// TwinCAT 3 PLC project MoldingCooler
// Title: Molding Cooling Tunnel
// Company: D_WFinePack
// ProjectVersion: 1.1.0
// ProgramVersion: 3.1.4020.4
// libraries:
//   Tc2_EtherCAT, * (Beckhoff Automation GmbH)
//   Tc2_Standard, * (Beckhoff Automation GmbH)
//   Tc2_System, * (Beckhoff Automation GmbH)
//   Tc2_SystemCX, * (Beckhoff Automation GmbH)
//   Tc2_Utilities, * (Beckhoff Automation GmbH)
//   Tc3_Module, * (Beckhoff Automation GmbH)
//   TemplateCore, * (TemplateCore Creators)
// project tree:
//   DUTs/Constants/ udtConstantsTransactions.TcDUT
//   DUTs/Database/ udtDBChannel.TcDUT, udtDBInterface.TcDUT, udtDBStoreFault.TcDUT, udtDBTransact.TcDUT
//   DUTs/RecipeData/ udtRecipe.TcDUT
//   DUTs/ udtCmpBaseMain.TcDUT, udtCmpServo.TcDUT, udtCmpVFD.TcDUT, udtEthercatSlaveStatus.TcDUT, udtHourlyData.TcDUT, udtIWS_DataLogItems.TcDUT, udtVFDCommand.TcDUT, udtVFDStatus.TcDUT, udtYaskawaVFDCmd.TcDUT, udtYaskawaVFDStatus.TcDUT
//   GVLs/ Globals.TcGVL
//   / PlcTask.TcTTO
//   POUs/ FB_DBTransaction.TcPOU, FB_PID.TcPOU, FB_Sensor.TcPOU, GlobalConfig.TcPOU, GlobalLogic.TcPOU
//   POUs/Stn100/ Stn100_00_ModeControl.TcPOU, Stn100_01_HMI.TcPOU, Stn100_02_Stats.TcPOU, Stn100_10_Main.TcPOU, Stn100_20_CoolingConveyor.TcPOU, Stn100_30_VibratoryConveyor.TcPOU, Stn100_40_Vibrator.TcPOU
// real-time tasks:
//   TASK PlcTask: cycle T#10ms, priority 10, ADS port 350
// I/O:
//   DEVICE EtherCat Master (EtherCAT), AmsNetId 5.49.24.194.2.1
//     Term 12 (EK1200) [EK1200-5000 EtherCAT Power supply (2A E-Bus)]
//       Term 13 (EL6070-0033) [EL6070-0033 1Ch. Licence key terminal, individual licences]
//       Term 14 (EL1034) [EL1034 4Ch. Dig. Input 24V, potential-free, 10µs]
//       Term 16 (EL1034) [EL1034 4Ch. Dig. Input 24V, potential-free, 10µs]
//       Term 17 (EL1034) [EL1034 4Ch. Dig. Input 24V, potential-free, 10µs]
//       Term 18 (EL1034) [EL1034 4Ch. Dig. Input 24V, potential-free, 10µs]
//       Term 19 (EL2798) [EL2798 8Ch. Dig. Output 24V AC/DC, 2A, potential-free]
//       Term 20 (EL2798) [EL2798 8Ch. Dig. Output 24V AC/DC, 2A, potential-free]
//       Term 21 (EL3314-0010) [EL3314-0010 4Ch. Ana Input Thermocouple (TC), High Precision]
//       Term 21 (EL6652) [EL6652 EtherNet/IP Scanner (Master)]
//       Term 23 (EK1110) [EK1110 EtherCAT extension]
//     Box 24 (Cooling Conv YASKAWA V1000 series) [YASKAWA V1000 series]
//     Box 25 (Vib Conv YASKAWA V1000 series) [YASKAWA V1000 series]
//     Box 26 (Vib Shaker YASKAWA V1000 series) [YASKAWA V1000 series]
//   DEVICE Device 2 (ECAT EIP Scanner (EL6652)), AmsNetId 5.49.24.194.3.1
//     Box 1 (FP7CPUS UNIT AFP7CPS31ES) // <INFO> </INFO> <EDS> 00D8000C00030100WN5.eds </EDS>
// variable links:
//   MoldingCooler/MoldingCooler Instance <-> Device 2 (ECAT EIP Scanner (EL6652))/Box 1 (FP7CPUS UNIT AFP7CPS31ES)
//     PlcTask Inputs/.gWeighRightCurrentRecipeID <-> Connection 2 (Input/Output)/Inputs/InByte_3
//     PlcTask Inputs/.gWeighRightInputs <-> Connection 2 (Input/Output)/Inputs/InByte
//   MoldingCooler/MoldingCooler Instance <-> EtherCat Master (EtherCAT)/Box 24 (Cooling Conv YASKAWA V1000 series)
//     PlcTask Inputs/Stn100_20_CoolingConveyor.iCurrentVelocity <-> Inputs_1/Output frequency
//     PlcTask Inputs/Stn100_20_CoolingConveyor.iStatus <-> Inputs/Drive status
//     PlcTask Outputs/Stn100_20_CoolingConveyor.oCommand <-> Outputs/Operation command
//     PlcTask Outputs/Stn100_20_CoolingConveyor.oSpeedReference <-> Outputs_1/Speed reference/limit
//   MoldingCooler/MoldingCooler Instance <-> EtherCat Master (EtherCAT)/Box 25 (Vib Conv YASKAWA V1000 series)
//     PlcTask Inputs/Stn100_30_VibratoryConveyor.iCurrentVelocity <-> Inputs_1/Output frequency
//     PlcTask Inputs/Stn100_30_VibratoryConveyor.iStatus <-> Inputs/Drive status
//     PlcTask Outputs/Stn100_30_VibratoryConveyor.oCommand <-> Outputs/Operation command
//     PlcTask Outputs/Stn100_30_VibratoryConveyor.oSpeedReference <-> Outputs_1/Speed reference/limit
//   MoldingCooler/MoldingCooler Instance <-> EtherCat Master (EtherCAT)/Box 26 (Vib Shaker YASKAWA V1000 series)
//     PlcTask Inputs/Stn100_40_Vibrator.iCurrentVelocity <-> Inputs_1/Output frequency
//     PlcTask Inputs/Stn100_40_Vibrator.iStatus <-> Inputs/Drive status
//     PlcTask Outputs/Stn100_40_Vibrator.oCommand <-> Outputs/Operation command
//     PlcTask Outputs/Stn100_40_Vibrator.oSpeedReference <-> Outputs_1/Speed reference/limit
//   MoldingCooler/MoldingCooler Instance <-> EtherCat Master (EtherCAT)/Term 12 (EK1200)/Term 14 (EL1034)
//     PlcTask Inputs/Stn100_00_ModeControl.iMovenCoolTankFull <-> Channel 2/Input
//     PlcTask Inputs/Stn100_10_Main.iBoxPres_Filling <-> Channel 4/Input
//     PlcTask Inputs/Stn100_10_Main.iWR_FillCmp <-> Channel 3/Input
//   MoldingCooler/MoldingCooler Instance <-> EtherCat Master (EtherCAT)/Term 12 (EK1200)/Term 16 (EL1034)
//     PlcTask Inputs/.iCycleStart <-> Channel 3/Input
//     PlcTask Inputs/.iCycleStop <-> Channel 4/Input
//   MoldingCooler/MoldingCooler Instance <-> EtherCat Master (EtherCAT)/Term 12 (EK1200)/Term 17 (EL1034)
//     PlcTask Inputs/Stn100_10_Main.iBoxPres_InfeedEntrance <-> Channel 1/Input
//     PlcTask Inputs/Stn100_10_Main.iBoxPres_Infeeed <-> Channel 2/Input
//     PlcTask Inputs/Stn100_10_Main.iBoxPres_OutFeed <-> Channel 3/Input
//     PlcTask Inputs/Stn100_10_Main.iBoxPres_OutFeedExit <-> Channel 4/Input
//   MoldingCooler/MoldingCooler Instance <-> EtherCat Master (EtherCAT)/Term 12 (EK1200)/Term 18 (EL1034)
//     PlcTask Inputs/Stn100_10_Main.iBoxCyl_DS_Retd <-> Channel 1/Input
//     PlcTask Inputs/Stn100_10_Main.iBoxCyl_US_Retd <-> Channel 2/Input
//   MoldingCooler/MoldingCooler Instance <-> EtherCat Master (EtherCAT)/Term 12 (EK1200)/Term 19 (EL2798)
//     PlcTask Outputs/Stn100_10_Main.oBoxCyl_DS_Ret <-> Channel 7/Output
//     PlcTask Outputs/Stn100_10_Main.oBoxCyl_US_Ret <-> Channel 8/Output
//     PlcTask Outputs/Stn100_10_Main.oInfeedConv_EntRelease <-> Channel 3/Output
//     PlcTask Outputs/Stn100_10_Main.oInfeedConv_Release <-> Channel 4/Output
//     PlcTask Outputs/Stn100_10_Main.oOutFeedConv_ExitRelease <-> Channel 6/Output
//     PlcTask Outputs/Stn100_10_Main.oOutFeedConv_Recieve <-> Channel 5/Output
//     PlcTask Outputs/Stn100_10_Main.oWeighRight_Ok2Fill <-> Channel 1/Output
//   MoldingCooler/MoldingCooler Instance <-> EtherCat Master (EtherCAT)/Term 12 (EK1200)/Term 20 (EL2798)
//     PlcTask Outputs/Stn100_00_ModeControl.oStackLightGreen <-> Channel 3/Output
//     PlcTask Outputs/Stn100_00_ModeControl.oStackLightHorn <-> Channel 4/Output
//     PlcTask Outputs/Stn100_00_ModeControl.oStackLightRed <-> Channel 1/Output
//     PlcTask Outputs/Stn100_00_ModeControl.oStackLightYellow <-> Channel 2/Output
//   MoldingCooler/MoldingCooler Instance <-> EtherCat Master (EtherCAT)/Term 12 (EK1200)/Term 21 (EL3314-0010)
//     PlcTask Inputs/Stn100_10_Main.iTempAtMoldDrop <-> TC Inputs Channel 1/Value
//     PlcTask Inputs/Stn100_10_Main.iTempAtShuteDrop <-> TC Inputs Channel 2/Value

CONFIGURATION MoldingCooler
    RESOURCE PLC ON TwinCAT3
        TASK PlcTask(INTERVAL := T#10ms, PRIORITY := 10);
        PROGRAM GlobalConfig WITH PlcTask : GlobalConfig;
        PROGRAM GlobalLogic WITH PlcTask : GlobalLogic;
        PROGRAM Stn100_00_ModeControl WITH PlcTask : Stn100_00_ModeControl;
        PROGRAM Stn100_01_HMI WITH PlcTask : Stn100_01_HMI;
        PROGRAM Stn100_02_Stats WITH PlcTask : Stn100_02_Stats;
        PROGRAM Stn100_10_Main WITH PlcTask : Stn100_10_Main;
        PROGRAM Stn100_20_CoolingConveyor WITH PlcTask : Stn100_20_CoolingConveyor;
        PROGRAM Stn100_30_VibratoryConveyor WITH PlcTask : Stn100_30_VibratoryConveyor;
        PROGRAM Stn100_40_Vibrator WITH PlcTask : Stn100_40_Vibrator;
    END_RESOURCE
END_CONFIGURATION

// ---- DUTs/Constants/udtConstantsTransactions.TcDUT
TYPE udtConstantsTransactions :
STRUCT
	FindSlot : INT := 1;
	GetAssignedStation: INT := 2;
	GetLineStatus : INT := 3;
	GetOrderData : INT := 4;
	GetPalletData: INT := 5;
	GetUnusedPalletID : INT := 6;
	SetOrderData : INT := 7;
	SetPalletData : INT := 8;
	StoreFault : INT := 9;
	GetAlignerData : INT := 10;
	DebugGetPartialAID : INT := 11;
	SetManualAID : INT :=12;
	DebugLookupAlignerInBatch :INT := 13;
	DebugAssignDummyAligner :INT := 14;
END_STRUCT
END_TYPE

// ---- DUTs/Database/udtDBChannel.TcDUT
TYPE udtDBChannel :
STRUCT
	CurrentUser:DINT;
	ErrorCode: DINT;
	ErrorMessage: STRING[256];
	DataIn: ARRAY[0..1999] OF BYTE;
	DataOut: ARRAY[0..1999] OF BYTE;
END_STRUCT
END_TYPE

// ---- DUTs/Database/udtDBInterface.TcDUT
TYPE udtDBInterface :
STRUCT
	Trigger: DWORD;
	Response: DWORD;
	Lock: BOOL;
	Connection: ARRAY[0..19] OF udtDBChannel;
END_STRUCT
END_TYPE

// ---- DUTs/Database/udtDBStoreFault.TcDUT
TYPE udtDBStoreFault :
STRUCT
	Station : DINT;
	FaultCode: DINT;
	FaultText : STRING[255];
	AcknowledgeTime: REAL;
	Duration: REAL;
	TimeStamp:Timestamp;
	Data1 : REAL;
	Data2 : REAL;
	Data3:  REAL;
	StringData1 : STRING[255];
	StringData2 : STRING[255];
	ResultCode: DINT;
	ResultText: STRING[255] ;
END_STRUCT
END_TYPE

// ---- DUTs/Database/udtDBTransact.TcDUT
TYPE udtDBTransact :
STRUCT
	Start: BOOL;
	Done: BOOL;
	ErrorCode: DINT;
	ErrorMessage : STRING[256];
	pDatabaseInterface: POINTER TO udtDBInterface;
	UserID: DINT;
	TransactionID: INT;
	DataLength: DINT;
	DataOutLength: DINT;
	DataIn: ARRAY[0..1999] OF BYTE;
	DataOut: ARRAY[0..1999] OF BYTE;
	State: DINT;
END_STRUCT
END_TYPE

// ---- DUTs/RecipeData/udtRecipe.TcDUT
TYPE udtRecipe :
STRUCT
	Matnr: STRING;
	Maktx: STRING;
	Pic_Name: STRING;
	VisionID: DINT;
	nBatchID: DINT;
	QuantityToProduce: DINT;
	Remaining: DINT;
	LoadConv_Speed: REAL;
	HopperElev_Speed: REAL;
	SeparatorConv_Speed: REAL;
	PaddleWheel_Speed: REAL;
	SortingConv_Speed: REAL;
	Wrapper_Speed: REAL;
	Wrapper_TempSP: REAL;
	Wrapper_VacuumSP: REAL;
END_STRUCT
END_TYPE

// ---- DUTs/udtCmpBaseMain.TcDUT
TYPE udtCmpBaseMain :
STRUCT
	Framework: Framework;
END_STRUCT
END_TYPE

// ---- DUTs/udtCmpServo.TcDUT
TYPE udtCmpServo :
STRUCT
	Framework: Framework;
	BaseSpeedRef: REAL;
	RunReq: BOOL;
	Running: BOOL;
END_STRUCT
END_TYPE

// ---- DUTs/udtCmpVFD.TcDUT
TYPE udtCmpVFD :
STRUCT
	Framework: Framework;
	BaseSpeedRef: REAL;
	RunReq: BOOL;
	Running: BOOL;
END_STRUCT
END_TYPE

// ---- DUTs/udtEthercatSlaveStatus.TcDUT
TYPE udtEthercatSlaveStatus :
STRUCT
	Address : WORD;
	Name : STRING[31];
	DeviceState: BYTE;
	LinkState: BYTE;
	SlaveStateBits: ST_EcSlaveStateBits;
END_STRUCT
END_TYPE

// ---- DUTs/udtHourlyData.TcDUT
TYPE udtHourlyData :
STRUCT
	GoodCount :DINT :=0;
	ScrapCount :DINT :=0;	
END_STRUCT
END_TYPE

// ---- DUTs/udtIWS_DataLogItems.TcDUT
TYPE udtIWS_DataLogItems :
STRUCT
	HourlyTranReq :BOOL  :=0;
	HourlyTranCmp :BOOL  :=0;
	CurrOeeTranReq :BOOL  :=0;
	CurrOeeTranCmp :BOOL  :=0;
	ShiftOeeTranReq :BOOL  :=0;
	ShiftOeeTranCmp :BOOL  :=0;
	FaultedTranReq :BOOL  :=0;
	FaultedTranCmp :BOOL  :=0;
	FailureTranReq :BOOL  :=0;
	FailureTranCmp :BOOL  :=0;
	CreateNewBatchReq :BOOL  :=0;
	CreateNewBatchCmp :BOOL  :=0;
END_STRUCT
END_TYPE

// ---- DUTs/udtVFDCommand.TcDUT
TYPE udtVFDCommand :
STRUCT
	Stop : BOOL;
	Start: BOOL;
	Jog: BOOL;
	ClearFaults: BOOL;
	RunFwd: BOOL;
	RunRev: BOOL;
	ForceKeypadCtrl: BOOL;
	MOPIncrement: BOOL;
	AccelRate1: BOOL;
	AccelRate2: BOOL;
	DecelRate1: BOOL;
	DecelRate2: BOOL;
	FreqSel01: BOOL;
	FreqSel02: BOOL;
	FreqSel03: BOOL;
	MOPDecrement: BOOL;
END_STRUCT
END_TYPE

// ---- DUTs/udtVFDStatus.TcDUT
TYPE udtVFDStatus :
STRUCT
	Ready : BOOL;
	Active: BOOL;
	CommandFwd: BOOL;
	RunningFwd: BOOL;
	Accelerating: BOOL;
	Decelerating: BOOL;
	Reserved: BOOL;	
	Faulted: BOOL;
	AtSpeed: BOOL;
	CommFreqCnt: BOOL;
	CommLogicCnt: BOOL;
	ParmsLocked: BOOL;
	DigIn1Active: BOOL;
	DigIn2Active: BOOL;
	DigIn3Active: BOOL;
	DigIn4Active: BOOL;
END_STRUCT
END_TYPE

// ---- DUTs/udtYaskawaVFDCmd.TcDUT
TYPE udtYaskawaVFDCmd :
STRUCT
	RunFwd :BOOL;
	RunRev :BOOL;
	ClearFaults :BOOL;	
END_STRUCT
END_TYPE

// ---- DUTs/udtYaskawaVFDStatus.TcDUT
TYPE udtYaskawaVFDStatus :
STRUCT
Running :BOOL;	
ZeroSpeed :BOOL;
RunningFWD :BOOL;
SpeedAgree :BOOL;
Ready :BOOL;
Alarm :BOOL;
Faulted :BOOL;
OpError :BOOL;
PowerLoss:BOOL;
END_STRUCT
END_TYPE

// ---- GVLs/Globals.TcGVL
{attribute 'Tc2GvlVarNames'}
{attribute 'qualified_only'}
VAR_GLOBAL
	(*Wired Inputs for Station Control*)
	iCycleStart AT %I* :BOOL;
	iCycleStop AT %I* :BOOL;
	
	gDatabaseInterface: udtDBInterface;
	gInitialScanForce: BOOL:=0;
	gFirstScan: BOOL:=0;
	gTimeZoneOffsetFromUTC: DINT;
	gCurrentTime: timestamp;
	gSoftwareRevision : STRING;
	gDbTransact :ARRAY[0..1] OF udtIWS_DataLogItems;
	
	(*Create the Hourly Containers*)
	gCurrShift :DINT;
	gLastShift :DINT;
	gCurrentHour :DINT;
	gLastHour : DINT;
	gTargetRatePerHour : DINT;
	gTargetRatePerMin : DINT;
	gRejectRate : REAL;
	gHourlyData: ARRAY[0..23] OF udtHourlyData;
	gShiftdata :ARRAY[0..3] OF udtHourlyData;
	gCurrOeeLogTime :TIME := T#300000MS;
	

	(*Station 100*)
	gStation100: Station;
	gStn100_02_Stats : Component_Stats;
	gStn100_StateTraceBuffer : TraceFIFOBuffer;
	gStn100_StateTraceFifo : FIFO_StateTrace := ( Overwrite := TRUE );
	gStn100_HMIMessageBuffer : HMIMessageBuffer;
	gStn100_HMIMessageFIFO : FIFO_HMIMessage := (Overwrite := TRUE);
	gStn100_10_Main : udtCmpBaseMain;
	gStn100_20_CoolingConveyor : udtCmpVFD;
	gStn100_30_VibratoryConveyor : udtCmpVFD;
	gStn100_40_Vibrator : udtCmpVFD;
	gStn100FaultedNotAck: BOOL;	
	
	(* Ethernet IP Inputs from Weigh Scale *)
		gWeighRightInputs AT %I* : INT;
		gWeighRightCurrentRecipeID AT %I* :INT;

END_VAR

VAR_GLOBAL PERSISTENT
	gCurrProduct : udtRecipe;
END_VAR

VAR_GLOBAL CONSTANT
	strNull : STRING :='';
	cStats: StatsConstants;
	gstLibVersion : ST_LibVersion;
END_VAR

// ---- POUs/GlobalConfig.TcPOU
PROGRAM GlobalConfig
VAR
	FirstScan:R_TRIG;
	FBStartHMI:NT_StartProcess;
	tmrDelayHMIStart:TON;

	fbNTGetLocalTime : FB_LocalSystemTime;
	LocalSystemTime : T_FileTime;
	fbDisplay : FB_CXSetTextDisplay;
	hiStartOfShift1Min : DINT;
	hiStartOfShift1Hour : DINT;
	hiStartOfShift2Min : DINT;
	hiStartOfShift2Hour : DINT;
	hiStartOfShift3Min : DINT;
	hiStartOfShift3Hour : DINT;
	hiPlannedDownTimeShift1Min : DINT;
	hiPlannedDownTimeShift2Min : DINT;
	hiPlannedDownTimeShift3Min : DINT;
	hiIdealCycleTime : REAL;
	hiAggregateInterval : DINT;
	TempFullRate : DINT;
	TempRateCalc : FLOAT;
	tempRejectRate : FLOAT;
	
	tTime : TimeStamp;
	END_VAR

FirstScan(CLK:=TRUE);
Globals.gFirstScan:=FirstScan.Q OR Globals.gInitialScanForce;
Globals.gInitialScanForce := FALSE;
IF Globals.gFirstScan THEN
	(*Initialize all FIFOs to avoid Access Violation exception*)
	Globals.gStn100_StateTraceFifo.INIT(pFIFO := ADR(Globals.gStn100_StateTraceBuffer));
	Globals.gStation100.AttentionRequiredFIFO.INIT(pFIFO := ADR(Globals.gStation100.AttentionRequiredFIFOBuffer));
	Globals.gStation100.NotOKtoStopFIFO.INIT(pFIFO := ADR(Globals.gStation100.NotOKToStopFIFOBuffer));
	Globals.gStation100.FaultedFIFO.INIT(pFIFO := ADR(Globals.gStation100.FaultedFIFOBuffer));
	Globals.gStation100.HMIMessageFIFO.INIT(pFIFO := ADR(Globals.gStation100.HMIMessageBuffer));
	
	(*Set Time Zone*)
	Globals.gTimeZoneOffsetFromUTC := -7;
	Globals.gSoftwareRevision := Dint_to_String(Globals.gstLibVersion.iRevision);
	Globals.gStation100.MachineID :=4;
	
	(*Set Initial Start Of Shift Values HackAlert*)
	Globals.gStn100_02_Stats.StartOfShift[0,0] :=0;	
	Globals.gStn100_02_Stats.StartOfShift[0,1] :=7;	
	Globals.gStn100_02_Stats.StartOfShift[1,0] :=0;	
	Globals.gStn100_02_Stats.StartOfShift[1,1] :=15;	
	Globals.gStn100_02_Stats.StartOfShift[2,0] :=0;	
	Globals.gStn100_02_Stats.StartOfShift[2,1] :=23;		
END_IF

(*Set display*)
fbDisplay(bExecute := Globals.gFirstScan,
			nDevID := 2,
			nMode := e_CX1100_WRITELine1,
			stLine := 'DW2164_rev01',
			nCursorPos := 0);

fbNTGetLocalTime(
	sNetID:='' ,
	bEnable:= TRUE,
	dwCycle:= 1,
	dwOpt:= 0,
	tTimeout:= DEFAULT_ADS_TIMEOUT );
LocalSystemTime := SYSTEMTIME_TO_FILETIME(fbNTGetLocalTime.systemTime);
Globals.gCurrentTime.CurrentValue.dwHighPart := LocalSystemTime.dwHighDateTime;
Globals.gCurrentTime.CurrentValue.dwLowPart := LocalSystemTime.dwLowDateTime;
Globals.gCurrentTime.DateTime := fbNTGetLocalTime.systemTime;
templatecore.GVL.gCurrentTime := Globals.gCurrentTime;

tTime := Globals.gCurrentTime;
tempRejectRate := (Globals.gRejectRate / 1000);
TempFullRate :=(Globals.gTargetRatePerMin*60);
TempRateCalc := FLOAT_TO_DINT(TempFullRate*(tempRejectRate));
Globals.gTargetRatePerHour := (TempFullRate-FLOAT_TO_DINT(TempRateCalc));

(*STATION 100*)
(*Reset logic for top-level main component*)
Globals.gStn100_10_Main.Framework.ResetStart := Globals.gStation100.CycleReset;
IF Globals.gStn100_10_Main.Framework.ResetDone THEN
	Globals.gStation100.ResetDone := TRUE;
ELSE
	Globals.gStation100.ResetDone := FALSE;
END_IF

(*Set Component IDs and Configurations*)
Globals.gStation100.StationID := 100;
Globals.gStn100_02_Stats.Framework.ComponentIDRecord.ID := 2;
Globals.gStn100_02_Stats.Framework.ComponentIDRecord.Name := 'Stats';
Globals.gStn100_10_Main.Framework.ComponentIDRecord.ID := 10;
Globals.gStn100_10_Main.Framework.ComponentIDRecord.Name := 'Main';
Globals.gStn100_20_CoolingConveyor.Framework.ComponentIDRecord.ID := 20;
Globals.gStn100_20_CoolingConveyor.Framework.ComponentIDRecord.Name := 'Cooling Conv';
Globals.gStn100_30_VibratoryConveyor.Framework.ComponentIDRecord.ID := 30;
Globals.gStn100_30_VibratoryConveyor.Framework.ComponentIDRecord.Name := 'Vibratory Conv';
Globals.gStn100_40_Vibrator.Framework.ComponentIDRecord.ID := 40;
Globals.gStn100_40_Vibrator.Framework.ComponentIDRecord.Name := 'Vibrator';


IF Globals.gStn100_02_Stats.IdealCycleTime <= 0.3 THEN
	Globals.gStn100_02_Stats.IdealCycleTime := 0.3; (*time in seconds*)
END_IF
Globals.gStn100_02_Stats.AggregateInterval := 3; (*aggregate time in minutes*)
IF Globals.gStn100_02_Stats.AggregateInterval < 1 THEN
	Globals.gStn100_02_Stats.AggregateInterval  := 1;
END_IF

(*Handle The HMI OEE Config Items*)
IF ((NOT Globals.gStation100.CycleAuto) AND (NOT Globals.gStation100.CycleFaulted)) THEN
	IF (hiStartOfShift1Min >0 AND hiStartOfShift1Min <> Globals.gStn100_02_Stats.StartOfShift[0,0]) THEN
		Globals.gStn100_02_Stats.StartOfShift[0,0] := hiStartOfShift1Min;
	END_IF
	IF (hiStartOfShift1Hour >0 AND hiStartOfShift1Hour <> Globals.gStn100_02_Stats.StartOfShift[0,1]) THEN
		Globals.gStn100_02_Stats.StartOfShift[0,1] := hiStartOfShift1Hour;
	END_IF
	IF (hiStartOfShift2Min >0 AND hiStartOfShift2Min <> Globals.gStn100_02_Stats.StartOfShift[1,0]) THEN
		Globals.gStn100_02_Stats.StartOfShift[1,0] := hiStartOfShift2Min;
	END_IF	
	IF (hiStartOfShift2Hour >0 AND hiStartOfShift2Hour <> Globals.gStn100_02_Stats.StartOfShift[1,1]) THEN
		Globals.gStn100_02_Stats.StartOfShift[1,1] := hiStartOfShift2Hour;
	END_IF	
	IF (hiStartOfShift3Min >0 AND hiStartOfShift3Min <> Globals.gStn100_02_Stats.StartOfShift[2,0]) THEN
		Globals.gStn100_02_Stats.StartOfShift[2,0] := hiStartOfShift3Min;
	END_IF	
	IF (hiStartOfShift3Hour >0 AND hiStartOfShift3Hour <> Globals.gStn100_02_Stats.StartOfShift[2,1]) THEN
		Globals.gStn100_02_Stats.StartOfShift[2,1] := hiStartOfShift3Hour;
	END_IF	
	IF (hiPlannedDownTimeShift1Min >0 AND hiPlannedDownTimeShift1Min <> Globals.gStn100_02_Stats.PlannedDownTime[0]) THEN
		Globals.gStn100_02_Stats.PlannedDownTime[0] := hiPlannedDownTimeShift1Min;
	END_IF	
	IF (hiPlannedDownTimeShift2Min >0 AND hiPlannedDownTimeShift2Min <> Globals.gStn100_02_Stats.PlannedDownTime[1]) THEN
		Globals.gStn100_02_Stats.PlannedDownTime[1] := hiPlannedDownTimeShift2Min;
	END_IF	
	IF (hiPlannedDownTimeShift3Min >0 AND hiPlannedDownTimeShift3Min <> Globals.gStn100_02_Stats.PlannedDownTime[2]) THEN
		Globals.gStn100_02_Stats.PlannedDownTime[2] := hiPlannedDownTimeShift3Min;
	END_IF		
	IF (hiIdealCycleTime >0 AND hiIdealCycleTime <> Globals.gStn100_02_Stats.IdealCycleTime) THEN
		Globals.gStn100_02_Stats.IdealCycleTime := hiIdealCycleTime;
	END_IF	
	IF (hiAggregateInterval >0 AND hiAggregateInterval <> Globals.gStn100_02_Stats.AggregateInterval) THEN
		Globals.gStn100_02_Stats.AggregateInterval := hiAggregateInterval;
	END_IF	
END_IF

END_PROGRAM

// ---- POUs/GlobalLogic.TcPOU
PROGRAM GlobalLogic
VAR
	(*Create the Objects for Data Collection of Rates*)
	hiHourDataLogReq :BOOL :=0;
	hoHourDataLogAck :BOOL :=0;	
	hiShiftDataLogReq :BOOL :=0;
	hoShiftDataLogAck :BOOL :=0;
	hiCurrOeeLogReq  :BOOL :=0;
	hoCurrOeeLogAck  :BOOL :=0;	
	hiShiftOeeLogReq  :BOOL :=0;
	hoShiftOeeLogAck  :BOOL :=0;		

	State :DINT :=0;
	NextState :DINT :=0;
	FirstEntry: BOOL;
	tmrState: TON;	
	tmrState20 :TON;
	tmrState40 :TON;
	tmrState50 :TON;
	tmrState70 :TON;
	tmrState80 :TON;
	tmrState100 :TON;
	tmrState110 :TON;
	tmrCurrOeeLog :TON;	
END_VAR

IF Globals.gFirstScan THEN
	tmrCurrOeeLog(in:=TRUE,pt:=Globals.gCurrOeeLogTime);
END_IF

(*Set HMI Flags for the Requested Data Log Event*)
IF (Globals.gCurrShift <> Globals.gLastShift) THEN
	hiShiftDataLogReq :=TRUE;	
END_IF

IF (Globals.gCurrentHour <> Globals.gLastHour) THEN
	hiHourDataLogReq :=TRUE;	
END_IF
tmrCurrOeeLog(in:=TRUE);
IF (tmrCurrOeeLog.Q) THEN	
	hiCurrOeeLogReq :=TRUE;
END_IF

IF NextState <> State THEN
	(*code: Log state change into buffer*)
	FirstEntry := TRUE;
	State := NextState;
ELSE
	FirstEntry := FALSE;
END_IF

IF FirstEntry THEN
	tmrState(IN:=FALSE);
	tmrState20(IN:=FALSE);
	tmrState40(IN:=FALSE);
	tmrState50(IN:=FALSE);
	tmrState70(IN:=FALSE);
	tmrState80(IN:=FALSE);	
	tmrState100(IN:=FALSE);
	tmrState110(IN:=FALSE);	
END_IF

CASE State OF
	
0:	(*Check If we have any Data logging Requests *)
		IF (hiHourDataLogReq)OR(Globals.gDbTransact[0].HourlyTranReq AND Globals.gDbTransact[0].HourlyTranCmp) THEN
			Globals.gDbTransact[0].HourlyTranReq := TRUE;
			NextState:=10;
		END_IF
		IF (hiShiftDataLogReq)OR (Globals.gDbTransact[0].ShiftOeeTranReq AND Globals.gDbTransact[0].ShiftOeeTranCmp) THEN
			Globals.gDbTransact[0].ShiftOeeTranReq := TRUE;
			NextState:=40;
		END_IF	
		IF (hiCurrOeeLogReq) THEN
			Globals.gDbTransact[0].CurrOeeTranReq := TRUE;
			NextState:=70;
		END_IF
(*		IF (hiShiftOeeLogReq) THEN
			Globals.gDbTransact[0].ShiftOeeTranReq := TRUE;			
			NextState:=100;
		END_IF *)

10:	(*Wait for confirmation from HMI For Hourly data Logging*)

	tmrState(IN:=TRUE, PT:=T#3.0S);
	hoHourDataLogAck := (Globals.gDbTransact[0].HourlyTranReq AND Globals.gDbTransact[0].HourlyTranCmp);
	IF hoHourDataLogAck THEN
		NextState:=20;
		Globals.gDbTransact[0].HourlyTranReq := FALSE;
		Globals.gDbTransact[0].HourlyTranCmp := FALSE;
	END_IF
	IF  tmrState.Q THEN
		hiHourDataLogReq := FALSE;
		hoHourDataLogAck := FALSE;
		Globals.gDbTransact[0].HourlyTranReq := FALSE;
		Globals.gDbTransact[0].HourlyTranCmp := FALSE;
		NextState:=0;
	END_IF

20:	(*Clear Hour DataLogging Events*)
	hoHourDataLogAck := (Globals.gDbTransact[0].HourlyTranReq AND Globals.gDbTransact[0].HourlyTranCmp);
	tmrState20(IN:=TRUE, PT:=T#3.0S);
	IF NOT hoHourDataLogAck AND NOT tmrState.Q THEN
		Globals.gLastHour := Globals.gCurrentHour ;
		Globals.gHourlyData[Globals.gCurrentHour].GoodCount :=0;
		Globals.gHourlyData[Globals.gCurrentHour].ScrapCount :=0;
		NextState:=0;		
	END_IF
	IF  tmrState20.Q THEN
		hiHourDataLogReq := TRUE;
		hoHourDataLogAck := FALSE;
		NextState:=0;
	END_IF
	
40:	(*Wait for confirmation from HMI For Shift data Logging*)
	hoShiftDataLogAck :=(Globals.gDbTransact[0].ShiftOeeTranReq AND Globals.gDbTransact[0].ShiftOeeTranCmp);
	tmrState40(IN:=TRUE, PT:=T#3.0S);
	IF hoShiftDataLogAck THEN
		NextState:=50;
		Globals.gDbTransact[0].ShiftOeeTranReq := FALSE;
		Globals.gDbTransact[0].ShiftOeeTranCmp := FALSE;
	END_IF
	IF  tmrState40.Q THEN
		hiShiftDataLogReq := FALSE;
		hoShiftDataLogAck := FALSE;
		NextState:=0;
	END_IF

50:	(*Clear Shift data Logging Event*)
	hoShiftDataLogAck :=(Globals.gDbTransact[0].ShiftOeeTranReq AND Globals.gDbTransact[0].ShiftOeeTranCmp);
	tmrState50(IN:=TRUE, PT:=T#3.0S);
	IF NOT hoHourDataLogAck THEN
		Globals.gLastShift := Globals.gCurrShift;
		(*Globals.gShiftData[Globals.gCurrShift].GoodCount :=0;
		Globals.gShiftData[Globals.gCurrShift].ScrapCount :=0;
		MEMSET(ADR(Stn100_02_Stats.DBShiftOeeRecord),0,SIZEOF(Stn100_02_Stats.DBShiftOeeRecord)); *)
		hiShiftOeeLogReq :=FALSE;			
		NextState:=0;	
	END_IF
	IF  tmrState50.Q THEN
		hiShiftDataLogReq := TRUE;
		hoShiftDataLogAck := FALSE;
		NextState:=0;
	END_IF	

70:	(*Wait for confirmation from HMI For Current OEE Data Logging*)
	hoCurrOeeLogAck :=(Globals.gDbTransact[0].CurrOeeTranReq AND Globals.gDbTransact[0].CurrOeeTranCmp);
	tmrState70(IN:=TRUE, PT:=T#3.0S);
	IF hoCurrOeeLogAck OR tmrState70.Q THEN
		NextState:=80;
		tmrCurrOeeLog(IN:=FALSE);
		Globals.gDbTransact[0].CurrOeeTranReq := FALSE;
		Globals.gDbTransact[0].CurrOeeTranCmp := FALSE;
	END_IF
	IF  tmrState70.Q THEN
		hiCurrOeeLogReq := FALSE;
		hoCurrOeeLogAck := FALSE;
		tmrCurrOeeLog(IN:=TRUE);		
		NextState:=0;
	END_IF

80:	(*Clear Current Oee Data Logging Event*)
	hoCurrOeeLogAck :=(Globals.gDbTransact[0].CurrOeeTranReq AND Globals.gDbTransact[0].CurrOeeTranCmp);
	tmrState80(IN:=TRUE, PT:=T#3.0S);
	IF NOT hoCurrOeeLogAck THEN
		NextState :=0;
	END_IF
	
	IF  tmrState80.Q THEN
		hiCurrOeeLogReq := TRUE;
		hoCurrOeeLogAck := FALSE;
		Globals.gDbTransact[0].CurrOeeTranReq := FALSE;
		Globals.gDbTransact[0].CurrOeeTranCmp := FALSE;
		NextState:=0;
	END_IF	
	
100: (*Wait for confirmation from HMI For Shift OEE Data Logging*)
	tmrState100(IN:=TRUE, PT:=T#3.0S);
	IF hoShiftOeeLogAck OR tmrState100.Q THEN
		NextState:=110;
	END_IF
	IF  tmrState100.Q THEN
		hiShiftOeeLogReq := FALSE;
		hoShiftOeeLogAck := FALSE;
		NextState:=0;
	END_IF

110: (*Clear*)
	tmrState110(IN:=TRUE, PT:=T#3.0S);
	IF NOT hoShiftOeeLogAck THEN
		NextState :=0;
	END_IF
	
	IF  tmrState110.Q THEN
		hiShiftOeeLogReq := FALSE;
		hoShiftOeeLogAck := FALSE;
		NextState:=0;
	END_IF		
	
END_CASE

END_PROGRAM

// ---- POUs/Stn100/Stn100_00_ModeControl.TcPOU
PROGRAM Stn100_00_ModeControl
VAR
	pStation: POINTER TO Station;
	pMain: POINTER TO udtCmpBaseMain;
	Local: FrameworkLocal;
	tmrDelayPCStart: TON;
	tmrWritePersistentData: TON;
	tmrWritePersistentDataPulse: TON;
	fbStartPC: NT_StartProcess;
	fbGetTime: GETSYSTEMTIME;
	fbWritePersistentData: FB_WritePersistentData;
	StationResetRequest: BOOL;
	MsgText: STRING256;
	AltMsgText: STRING256;
	FaultText: STRING256;
	FaultAltText: STRING256;
	FaultNumber: INT;
	FaultData: StatsFault;
	StationLevelFault: BOOL;
	TempEvent: StatsEvent;
	TimeStamp: StateTimeStamp;
	CurrentTime: TIMESTRUCT;
	TimeLo: UDINT;
	TimeHi: UDINT;
	cmdStart: BOOL;
	cmdOperatorStop: BOOL;
	cmdMachineStop: BOOL;
	cmdFaultAcknowledge: BOOL;
	cmdFullInit: BOOL;
	cmdFaultReset: BOOL;
	cmdSingleStepOn: BOOL;
	cmdSingleStepOff: BOOL;
	cmdSingleStepAdvance: BOOL;
	cmdManualMode: BOOL;
	OKToStart: BOOL;
	OKToReset: BOOL;
	onsStart: R_TRIG;
	onsOperatorStop: R_TRIG;
	onsMachineStop: R_TRIG;
	onsFaultAcknowledge: R_TRIG;
	onsStationReset: R_TRIG;
	onsFaultReset: R_TRIG;
	onsSingleStepOn: R_TRIG;
	onsSingleStepOff: R_TRIG;
	onsSingleStepAdvance: R_TRIG;
	onsManualMode: R_TRIG;
	onsEStopNotOKHMIMessage: BOOL;
	onsEStopNotOKStartAttmpt: BOOL;
	onsPowerOnAttmpt: BOOL;
	onsAirNotOKHMIMessage: BOOL;
	onsAirNotOKStartAttempt: BOOL;
	onsEStopSafetyEDMErrorHMIMessage: BOOL;
	onsEStopSafetyEDMErrorStartAttempt: BOOL;
	onsGateSafetyEDMErrorHMIMessage: BOOL;
	onsGateSafetyEDMErrorStartAttempt: BOOL;
	onsSortingConvSafetyEDMErrorHMIMessage: BOOL;
	onsSortingConvSafetyEDMErrorStartAttempt: BOOL;
	onsCrossConvSafetyEDMErrorHMIMessage: BOOL;
	onsCrossConvSafetyEDMErrorStartAttempt: BOOL;	
	onsGateNotLockedHMIMessage: BOOL;
	onsPrematureStartAttempt: BOOL;
	onsStartAttemptBeforePreheat: BOOL;
	WaitForResetMsg: BOOL;
	SeparateAckAndReset: BOOL := TRUE;
	bStartingToRun: BOOL;
	b500msPulse: BOOL;
	tmrPulseON: TON;
	tmrPulseOFF: TON;
	tmrState: TON;
	tmrControlPowerPBPressedDelay: TON;
	tmrAirPressureNotOK: TON;
	tmrMoveNCoolTankNotOK: TON;
	tmrOKToStop: TON;
	tmrGateLock: TON;
	cColor: Colors;
	cChannel: Channels;
	cStats: StatsConstants;	
	
	(*Inputs*)
	iEStopOK :BOOL;
	iEStopGateOK: BOOL;
	iEstopMainEnclosurePBReleased: BOOL;
	iEstopGatePBReleased: BOOL;
	iEstopRobotPBReleased: BOOL;
	iEstopGateClosed: BOOL;
	iEstopWrapperPBReleased: BOOL;
	iEstopWrapperGateClosed: BOOL;
	iEStopSafetyEDMError: BOOL;
	iEStopGateSafetyEDMError: BOOL;
	iSortingConveyorSafetyEDMError: BOOL;
	iCrossConveyorSafetyEDMError: BOOL;
	iControlPowerOnPB AT %I*  : BOOL;
	iGateResetPB AT %I*  : BOOL;
	iGateLocked AT %I*  : BOOL;
	// iAirSupplyOK AT %I* : BOOL;
	iWeighRightEStop : BOOL;
	iAirSupplyOK: BOOL;
	iMovenCoolTankFull AT %I*: BOOL;

	(*Outputs*)
	oControlPowerReset: BOOL;
	oControlPowerOnPBLT AT %Q* : BOOL;
	oGateResetPBLT AT %Q* : BOOL;	
	oGateLock AT %Q* : BOOL;
	oStackLightRed AT %Q* : BOOL;
	oStackLightYellow AT %Q* : BOOL;	
	oStackLightGreen AT %Q* : BOOL;
	oStackLightHorn AT %Q* : BOOL;

	(*Operator Inputs*)
	hiGateLock: BOOL;
	hiGateUnlock: BOOL;
	hiTestIndicatorTree: BOOL;
	hiStationDryCycleEnable: BOOL;
	
	(*Operator Outputs*)
	hoCurrentStateModeControl: DINT;
	hoSingleStepEnabled: BOOL := FALSE; 
	hoStationDryCycleEnabled: BOOL := FALSE;
	hoFirstScan: BOOL;
END_VAR

IF Globals.gFirstScan THEN
	hoFirstScan := TRUE;
    FaultNumber := 1;
    FaultText := 'PLC changed from Program to Run';
	FaultAltText := 'No Alt Text';
    Local.State := 9999; (*Necessary to get state 0 to execute FirstEntry logic*)
    Local.NextState := 0;
	pStation := ADR(Globals.gStation100);
	pMain := ADR(Globals.gStn100_10_Main);	
	
	Local.pStateTraceBuffer := ADR(Globals.gStn100_StateTraceBuffer);
	Local.pStateTraceFifo := ADR(Globals.gStn100_StateTraceFifo);
	Local.pStats := ADR(Globals.gStn100_02_Stats);
END_IF

(*Delay PC Start*) (*Is this doing anything? If not, delete? JECDebug*)
IF Globals.gFirstScan THEN
	tmrDelayPCStart(IN:=FALSE);
	fbStartPC(START:=FALSE);
ELSE
	tmrDelayPCStart(IN:=TRUE,PT:=T#30S);
END_IF

(*Write persistent data every 10 seconds to insure data is retained*)
tmrWritePersistentData(IN := NOT tmrWritePersistentDataPulse.Q, PT := T#10S);
tmrWritePersistentDataPulse(IN := tmrWritePersistentData.Q, PT := T#2S);
fbWritePersistentData(PORT := 851, START := tmrWritePersistentData.Q, TMOUT := T#5S, MODE := 0);

(*Map Safety IO*)
iEStopOK := 1;
iAirSupplyOK :=1;
(* Map WeighRight EStop*)
iWeighRightEStop := Globals.gWeighRightInputs.3;

(*Copy time components to local tag for display on HMI*)
CurrentTime.wDay := Globals.gCurrentTime.DateTime.wDay;
CurrentTime.wDayOfWeek := Globals.gCurrentTime.DateTime.wDayOfWeek;
CurrentTime.wHour := Globals.gCurrentTime.DateTime.wHour;
CurrentTime.wMilliseconds := Globals.gCurrentTime.DateTime.wMilliseconds;
CurrentTime.wMinute := Globals.gCurrentTime.DateTime.wMinute;
CurrentTime.wMonth := Globals.gCurrentTime.DateTime.wMonth;
CurrentTime.wSecond := Globals.gCurrentTime.DateTime.wSecond;
CurrentTime.wYear := Globals.gCurrentTime.DateTime.wYear;

(*Call Input routine*)
Input();

(*Status from each component*)
pStation^.CycleFaulted := pStation^.FaultedFIFO.Count > 0 OR StationLevelFault;
pStation^.CycleManual := pStation^.CycleManualFIFO.Count > 0;
pStation^.Attention := pStation^.AttentionRequiredFIFO.Count > 0;
pStation^.OKToStop := FALSE;
IF (pStation^.NotOKtoStopFIFO.Count = 0) THEN
	tmrOKToStop(IN := TRUE, PT:=T#1.0S);
	IF tmrOKToStop.Q THEN
	    pStation^.OKToStop := TRUE;
	END_IF;
ELSE
    tmrOKToStop(IN := FALSE);
END_IF

(*Check for need of full initialization*)
IF cmdFullInit OR cmdManualMode OR Globals.gFirstScan THEN
	pStation^.FullInitRequired := TRUE;
END_IF

(*Station permissives*)
pStation^.OKForManual := NOT pStation^.CycleAuto AND NOT pStation^.CycleReset AND NOT pStation^.EmergencyStop AND pStation^.FullInitRequired;
// OKToReset := NOT pStation^.EmergencyStop AND iAirSupplyOK AND NOT pStation^.CycleManual;
// OKToStart := NOT pStation^.EmergencyStop AND iAirSupplyOK AND NOT pStation^.CycleFaulted AND NOT pStation^.CycleManual;
OKToReset := NOT pStation^.EmergencyStop AND NOT pStation^.CycleManual;
OKToStart := NOT pStation^.EmergencyStop AND NOT pStation^.CycleFaulted AND NOT pStation^.CycleManual;
(*Single Step*)
IF cmdSingleStepOn THEN
	pStation^.SingleStep := 1;
	hoSingleStepEnabled:=TRUE;
ELSIF pStation^.SingleStep AND (cmdSingleStepOff OR Globals.gFirstScan) THEN
	pStation^.SingleStep :=0;
	hoSingleStepEnabled:=FALSE;
END_IF
pStation^.StepAdvance:=pStation^.SingleStep AND cmdSingleStepAdvance;

(*Copy state to local for display on HMI*)
hoCurrentStateModeControl:=Local.State;

(*Mode Logic*)
IF Local.NextState <> Local.State THEN
	Local.FirstEntry := TRUE;
	Local.State := Local.NextState;
	fbGetTime(timeLoDW=>TimeStamp.TimeLo, timeHiDW=>TimeStamp.TimeHi);
	TimeStamp.ID := 0;
	TimeStamp.State := Local.State;
	Local.pStateTraceFifo^.INSERT(pFIFO := Local.pStateTraceBuffer, in := TimeStamp);
	tmrState(IN:=FALSE); (*clear timer if state changes*)
ELSE
	Local.FirstEntry := FALSE;
END_IF

CASE Local.State OF

0:	(*Faulted, Not Acknowledged*)
	IF  Local.FirstEntry THEN
		pStation^.CycleAuto := FALSE;
		pStation^.CycleReset := FALSE;
		pStation^.CycleManual := FALSE;
		(*Log fault event*)
		TempEvent.TimeStamp := Globals.gCurrentTime;
		TempEvent.EType := Globals.cStats.Faulted;
		TempEvent.Data[0] := DINT_TO_REAL(pStation^.FirstFault.FaultID);
		TempEvent.StringData[0] := pStation^.FirstFault.StringData[0];
		F_SendEvent(ADR(Local.pStats^.StatsEventFIFO), ADR(Local.pStats^.StatsEventBuffer), ADR(TempEvent));
	END_IF

	IF cmdFaultAcknowledge OR NOT SeparateAckAndReset THEN
		Local.NextState :=10;
	END_IF

10:	(*Faulted, Acknowledged*)
	IF   Local.FirstEntry THEN
		IF SeparateAckAndReset THEN
			(*Send event fault acknowledge*)
			TempEvent.EType := Globals.cStats.FaultAcknowledge;
			F_SendEvent (ADR(Local.pStats^.StatsEventFIFO ), ADR(Local.pStats^.StatsEventBuffer), ADR(TempEvent));
			pStation^.StationMessage.Text :='Fault Acknowledged';
			pStation^.StationMessage.AltText :='Error reconocido';
			pStation^.StationMessage.Color := cColor.Grey;
			F_AddMessage(pStation, 'Fault Acknowledged', '', cColor.Grey, cChannel.General);
		END_IF
		WaitForResetMsg := TRUE;
	END_IF

	IF OKToReset  THEN
		IF WaitForResetMsg AND SeparateAckAndReset  THEN
			WaitForResetMsg := FALSE;
			IF pStation^.FullInitRequired THEN
				MsgText := 'FULL INITIALIZATION REQUIRED.  Waiting for Station Reset';
			ELSE
				MsgText := 'Waiting for Station or Fault Reset';
			END_IF
			AltMsgText := 'Esperando confirmación de estación o falla';
			pStation^.StationMessage.Text :=MsgText;
			pStation^.StationMessage.AltText :=AltMsgText;
			pStation^.StationMessage.Color := cColor.Grey;
			F_AddMessage(pStation, MsgText, AltMsgText, cColor.Grey, cChannel.General);
		END_IF
		IF  (cmdFaultReset AND NOT pStation^.FullInitRequired) OR cmdFullInit  THEN
			Local.NextState := 20;
			pStation^.SingleStep :=0;
		END_IF
	END_IF

20:	(*Unlatch Faults - Fault/Station Reset*)
	IF  Local.FirstEntry THEN
		pStation^.UnlatchFaults := TRUE;
		IF NOT SeparateAckAndReset THEN
			(*Send event fault acknowledge*)
			TempEvent.EType := Globals.cStats.FaultAcknowledge;
			F_SendEvent (ADR(Local.pStats^.StatsEventFIFO ), ADR(Local.pStats^.StatsEventBuffer), ADR(TempEvent));
		END_IF
	END_IF

	IF NOT pStation^.CycleFaulted AND NOT StationLevelFault THEN
		pStation^.UnlatchFaults := FALSE;		
		IF NOT pStation^.FullInitRequired THEN
			Local.NextState := 30;
		ELSE
			Local.NextState := 60;
		END_IF
	END_IF

30:	(*Fault Reset*)
	IF  Local.FirstEntry THEN
		pStation^.CycleReset := TRUE;
		MEMSET(ADR(pStation^.FirstFault),0,SIZEOF(pStation^.FirstFault)); (*clear first fault*)
		MsgText := 'Resetting...';
		AltMsgText := 'Alt: Restablecimiento...';
		pStation^.StationMessage.Text :=MsgText;
		pStation^.StationMessage.AltText :=AltMsgText;
		pStation^.StationMessage.Color := cColor.Green;
		F_AddMessage(pStation, MsgText, AltMsgText, cColor.Green, cChannel.General);
	END_IF

	IF  pStation^.ResetDone AND NOT pStation^.CycleFaulted THEN
		pStation^.CycleReset := FALSE;
		Local.NextState := 100;
	END_IF
	IF pStation^.CycleFaulted OR cmdFullInit THEN
		pStation^.CycleReset := FALSE;
		Local.NextState:= 0;
	END_IF

60:	(*Station Reset*)
	IF  Local.FirstEntry THEN
		pStation^.CycleReset := TRUE;
		MEMSET(ADR(pStation^.FirstFault),0,SIZEOF(pStation^.FirstFault)); (*clear first fault*)
		MsgText := 'Resetting...';
		AltMsgText := 'Alt: Restablecimiento...';
		pStation^.StationMessage.Text :=MsgText;
		pStation^.StationMessage.AltText :=AltMsgText;
		pStation^.StationMessage.Color := cColor.Green;
		F_AddMessage(pStation, MsgText, AltMsgText, cColor.Green, cChannel.General);
		TempEvent.EType := Globals.cStats.Initialize;
		F_SendEvent (ADR(Local.pStats^.StatsEventFIFO ), ADR(Local.pStats^.StatsEventBuffer), ADR(TempEvent));
	END_IF

	IF  pStation^.ResetDone AND NOT pStation^.CycleFaulted THEN
		pStation^.CycleReset := FALSE;
		pStation^.FullInitRequired := FALSE;
		Local.NextState := 100;
	END_IF
	IF pStation^.CycleFaulted  THEN
		pStation^.CycleReset := FALSE;
		Local.NextState:= 0;
	END_IF

100:	(*Idle*)
	IF  Local.FirstEntry THEN
		pStation^.StopRequest := FALSE;
		StationResetRequest := FALSE;
		TempEvent.EType := Globals.cStats.CycleTime;
		TempEvent.Data[0]  := 1; (*cancel any incomplete cycle time*)
		F_SendEvent (ADR(Local.pStats^.StatsEventFIFO ), ADR(Local.pStats^.StatsEventBuffer), ADR(TempEvent));
		(*Stack light flash green*)
		MsgText := 'Idle';
		AltMsgText := 'Ocioso';
		pStation^.StationMessage.Text :=MsgText;
		pStation^.StationMessage.AltText :=AltMsgText;
		pStation^.StationMessage.Color := cColor.Grey;
		F_AddMessage(pStation, MsgText, AltMsgText, cColor.Grey, cChannel.General);
	END_IF

	IF cmdStart AND OKToStart AND NOT pStation^.FullInitRequired THEN
		bStartingToRun:=TRUE;
		Local.NextState :=200;
	END_IF
	IF pStation^.CycleFaulted THEN
		Local.NextState :=0;
	END_IF
	IF cmdFullInit AND OKToReset THEN
		Local.NextState :=60;
	END_IF

200:	(*Running*)
	IF  Local.FirstEntry THEN
		pStation^.CycleAuto := TRUE;
		bStartingToRun:=FALSE;
		(*Stack light green*)
		MsgText := 'Running';
		AltMsgText := 'Running';
		pStation^.StationMessage.Text :=MsgText;
		pStation^.StationMessage.AltText :=AltMsgText;
		pStation^.StationMessage.Color := cColor.Green;
		F_AddMessage(pStation, MsgText, AltMsgText, cColor.Green, cChannel.General);
		(*Send Working event*)
		TempEvent.EType := Globals.cStats.Working;
		F_SendEvent (ADR(Local.pStats^.StatsEventFIFO ), ADR(Local.pStats^.StatsEventBuffer), ADR(TempEvent));
	END_IF
	IF cmdOperatorStop THEN
		Local.NextState :=210;
	END_IF
	IF pStation^.CycleFaulted OR cmdMachineStop  THEN
		Local.NextState :=220;
	END_IF

210:	(*Operator Stop Requested. Machine stopping*)
	IF  Local.FirstEntry THEN
		pStation^.StopRequest := TRUE;
		(*Start button flash green*)
		MsgText := 'Stopping...';
		AltMsgText := 'Alt: Parada...';
		pStation^.StationMessage.Text :=MsgText;
		pStation^.StationMessage.AltText :=AltMsgText;
		pStation^.StationMessage.Color := cColor.Green;
		F_AddMessage(pStation, MsgText, AltMsgText, cColor.Green, cChannel.General);
		TempEvent.EType := Globals.cStats.CycleTime;
		TempEvent.Data[0] := 1; (*cancel cycle timer*)
		F_SendEvent (ADR(Local.pStats^.StatsEventFIFO ), ADR(Local.pStats^.StatsEventBuffer), ADR(TempEvent));
	END_IF

	IF pStation^.OKToStop  THEN
		pStation^.CycleAuto := FALSE;
		IF pStation^.CycleFaulted THEN
			Local.NextState :=0;
		ELSE
			TempEvent.EType := Globals.cStats.OperatorStop;
			F_SendEvent (ADR(Local.pStats^.StatsEventFIFO ), ADR(Local.pStats^.StatsEventBuffer), ADR(TempEvent));
			Local.NextState := 100;
		END_IF
	END_IF

220:	(*Machine Stop Requested, or machine fault.. Machine stopping*)
	IF  Local.FirstEntry THEN
		pStation^.StopRequest := TRUE;
		(*Start button flash green*)
		TempEvent.EType := Globals.cStats.CycleTime;
		TempEvent.Data[0] := 1; (*cancel cycle timer*)
		F_SendEvent (ADR(Local.pStats^.StatsEventFIFO ), ADR(Local.pStats^.StatsEventBuffer), ADR(TempEvent));
	END_IF

	IF pStation^.OKToStop  THEN
		pStation^.CycleAuto := FALSE;
		IF pStation^.CycleFaulted   THEN
			Local.NextState :=0;
		ELSE
			TempEvent.EType := Globals.cStats.MachineStop;
			F_SendEvent (ADR(Local.pStats^.StatsEventFIFO ), ADR(Local.pStats^.StatsEventBuffer), ADR(TempEvent));
			Local.NextState := 100;
		END_IF
	END_IF
END_CASE

(*When a Control Power On PB is pressed, a Control Power Reset signal is sent to the Safety PLC.
  We delay before turning this signal off and checking for fault conditions.*)
tmrControlPowerPBPressedDelay(IN := (iControlPowerOnPB OR iGateResetPB OR 
								((tmrControlPowerPBPressedDelay.ET > T#0MS) AND NOT tmrControlPowerPBPressedDelay.Q)), PT := T#1000MS);
IF (tmrControlPowerPBPressedDelay.ET > T#0MS) AND (tmrControlPowerPBPressedDelay.ET < T#500MS) THEN
	oControlPowerReset := 1;
ELSE
	oControlPowerReset := 0;
END_IF

(*Station Level Fault Logic*)
(*Main Estop Relay and Doors*)
IF pStation^.EmergencyStop  THEN
	IF onsEStopNotOKHMIMessage THEN
		onsEStopNotOKHMIMessage := FALSE;
		FaultNumber := 2;
		FaultText := 'Emergency Stop';
		FaultAltText := 'Alt: Parada de emergencia';

		IF NOT iEstopMainEnclosurePBReleased AND NOT iWeighRightEStop THEN
			FaultNumber := 4;
			FaultText := CONCAT(FaultText, ' -Main Enclosure EStop PB pressed');
			FaultAltText := 'No Alt Text';
		END_IF
		IF iWeighRightEStop THEN
			FaultNumber := 14;
			FaultText := CONCAT(FaultText, ' -WeighRight EStop PB pressed');
			FaultAltText := 'No Alt Text';
		END_IF

	END_IF

	IF cmdStart OR cmdFaultReset OR cmdFullInit OR tmrControlPowerPBPressedDelay.Q THEN
		IF onsEStopNotOKStartAttmpt THEN
			onsEStopNotOKStartAttmpt := FALSE;			
			IF NOT iEStopOK THEN 
				MsgText := 'RESET or START attempted while EStops NOT Ok';
				AltMsgText := 'Alt: RESET o START intentado con la potencia de control no habilitada';
			ELSE
				onsPowerOnAttmpt := TRUE;;
			END_IF

			IF NOT iEstopMainEnclosurePBReleased THEN
				MsgText := 'RESET or START attempted while Main Enclosure ESTOP PB pressed';
				AltMsgText := 'Alt: Cabina de control Botón ESTOP presionado';
			END_IF
			IF iMovenCoolTankFull THEN
				MsgText := 'RESET or START attempted while Move N Coole Tank Full..';
				AltMsgText := 'Alt: ';			
			END_IF
			F_AddMessage(pStation, MsgText, AltMsgText, cColor.Red, cChannel.Attention);
		END_IF
	ELSE
		onsEStopNotOKStartAttmpt := TRUE;
		onsPowerOnAttmpt := FALSE;
	END_IF

ELSE
	IF onsPowerOnAttmpt THEN
		MsgText := ' ';
		AltMsgText := ' ';
		F_AddMessage(pStation, MsgText, AltMsgText, cColor.Grey, cChannel.General);
	END_IF
	onsEStopNotOKStartAttmpt := TRUE;
	onsEStopNotOKHMIMessage := TRUE;
	onsPowerOnAttmpt := FALSE;
END_IF

(*Main Air*)
IF NOT pStation^.EmergencyStop THEN // AND NOT iAirSupplyOK THEN
// tmrAirPressureNotOK(IN := pStation^.CycleAuto OR pStation^.CycleReset OR pStation^.CycleManual, PT := T#3.0s);
//	IF tmrAirPressureNotOK.Q THEN
//		IF onsAirNotOKHMIMessage THEN
//			onsAirNotOKHMIMessage := FALSE;
//			FaultNumber := 8;
//			FaultText := 'Air pressure NOT Ok';
//			FaultAltText := 'Alt: Pérdida de la presión de aire de la estación';
//		END_IF
//	ELSE
//		onsAirNotOKHMIMessage := TRUE;
//	END_IF
IF iMovenCoolTankFull THEN
	tmrMoveNCoolTankNotOK(IN := pStation^.CycleAuto OR pStation^.CycleReset OR pStation^.CycleManual, PT := T#2.0S);
	FaultNumber := 15;
	MsgText := 'START attempted with Move And Cool Tank Full or Not Present..';
	AltMsgText := 'Atl: START intentado con pérdida de presión de aire';
	F_AddMessage(pStation, MsgText, AltMsgText, cColor.Yellow, cChannel.Attention);
END_IF
	IF cmdStart OR cmdFaultReset OR cmdFullInit THEN
		IF onsAirNotOKStartAttempt THEN
			onsAirNotOKStartAttempt := FALSE;
			MsgText := 'START attempted with loss of air pressure';
			AltMsgText := 'Atl: START intentado con pérdida de presión de aire';
			F_AddMessage(pStation, MsgText, AltMsgText, cColor.Red, cChannel.Attention);
		END_IF
	ELSE
		onsAirNotOKStartAttempt := TRUE;
	END_IF
ELSE
	onsAirNotOKHMIMessage := TRUE;
	onsAirNotOKStartAttempt := TRUE;
	tmrAirPressureNotOK(IN := FALSE);
END_IF

(*EStop Safety EDM Error*) // if applicable Device attached
//IF iEStopSafetyEDMError THEN
//	IF onsEStopSafetyEDMErrorHMIMessage THEN
//		onsEStopSafetyEDMErrorHMIMessage := FALSE;
//		FaultNumber := 9;
//		FaultText := 'EStop safety EDM Error - check safety circuit';
//		FaultAltText := 'No Alt Text';
//	END_IF
//
//	IF cmdStart OR cmdFaultReset OR cmdFullInit OR tmrControlPowerPBPressedDelay.Q THEN
//		IF onsEStopSafetyEDMErrorStartAttempt THEN
//			onsEStopSafetyEDMErrorStartAttempt := FALSE;
//			MsgText := 'START attempted with EStop safety EDM Error - check safety circuit';
//			AltMsgText := 'No Alt Text';
//			F_AddMessage(pStation, MsgText, AltMsgText, cColor.Yellow, cChannel.Attention);
//		END_IF
//	ELSE
//		onsEStopSafetyEDMErrorStartAttempt := TRUE;
//	END_IF
//ELSE
//	onsEStopSafetyEDMErrorHMIMessage := TRUE;
//	onsEStopSafetyEDMErrorStartAttempt := TRUE;
//END_IF

(*Post station level fault*)
IF FaultNumber <> 0 AND  NOT StationLevelFault THEN
	StationLevelFault := TRUE;
	FaultData.FaultID := FaultNumber;
	FaultData.TimeStamp := Globals.gCurrentTime;
	MsgText :=  'Fault: ';
	AltMsgText  := 'AltFault: ';
	MsgText := CONCAT(MsgText,DINT_TO_STRING(FaultData.FaultID));
	MsgText := CONCAT(MsgText,' ');
	MsgText := CONCAT(MsgText, FaultText);
	AltMsgText := CONCAT(AltMsgText,DINT_TO_STRING(FaultData.FaultID));
	AltMsgText := CONCAT(AltMsgText,' ');
	AltMsgText:=CONCAT(AltMsgText, FaultAltText);
	F_AddMessage(pStation, MsgText, AltMsgText, cColor.Red, cChannel.Fault);
	IF pStation^.FirstFault.FaultID = 0 THEN
		pStation^.FirstFault := FaultData;
		pStation^.FirstFault.StationID  := pStation^.StationID;
		pStation^.FirstFault.StringData[0] :=MsgText;
		pStation^.FirstFault.StringData[1] :=AltMsgText;
	END_IF
END_IF

IF pStation^.UnlatchFaults THEN
	FaultNumber := 0;
	StationLevelFault := FALSE;
END_IF

(*Outputs*)
IF (pStation^.CycleFaulted AND b500msPulse) OR hiTestIndicatorTree THEN
	oStackLightRed := TRUE;
ELSIF oStackLightRed THEN
	oStackLightRed := FALSE;
END_IF

IF (NOT pStation^.CycleFaulted AND (pStation^.CycleAuto OR (NOT pStation^.CycleAuto AND b500msPulse))) 
  OR hiTestIndicatorTree THEN
	oStackLightGreen := TRUE;
ELSIF oStackLightGreen THEN
	oStackLightGreen := FALSE;
END_IF

IF (pStation^.Attention AND b500msPulse) OR hiTestIndicatorTree THEN
	oStackLightYellow := TRUE;
ELSIF oStackLightYellow THEN
	oStackLightYellow := FALSE;
END_IF

IF ((Local.State = 0) AND b500msPulse) OR hiTestIndicatorTree THEN
	oStackLightHorn := TRUE;
ELSIF oStackLightHorn THEN
	oStackLightHorn := FALSE;
END_IF

(*Turn on the Control Power On lights if Control Power is On, system air pressure is ok, and there are no safety EDM errors*)
IF (iEStopOK AND iAirSupplyOK AND NOT iEStopSafetyEDMError AND NOT iEStopGateSafetyEDMError 
  AND NOT iSortingConveyorSafetyEDMError) OR hiTestIndicatorTree THEN
	IF iEStopGateOK OR b500msPulse THEN
		oControlPowerOnPBLT := 1;
		oGateResetPBLT := 1;
	ELSE
		oControlPowerOnPBLT := 0;
		oGateResetPBLT := 0;
	END_IF
ELSE
	oControlPowerOnPBLT := 0;
	oGateResetPBLT := 0;	
END_IF

Globals.gStn100FaultedNotAck := Local.State = 0;

hoStationDryCycleEnabled := hiStationDryCycleEnable;
pStation^.DryCycle := hiStationDryCycleEnable;
pStation^.EmergencyStop := NOT iEStopOK OR iWeighRightEStop;

IF (pStation^.CycleAuto OR pStation^.CycleReset OR bStartingToRun) AND NOT pStation^.EmergencyStop THEN
	oGateLock := TRUE;
ELSIF pStation^.OKForManual THEN	(*Manual operation*)
	IF hiGateLock THEN
		oGateLock:=TRUE;
	END_IF
	IF hiGateUnlock THEN
		oGateLock:=FALSE;
	END_IF
ELSIF oGateLock THEN
	oGateLock := FALSE;
END_IF

(*1/2 second pulse generator*)
tmrPulseON(IN:=NOT tmrPulseOFF.Q,PT:=T#0.5s);
tmrPulseOFF(IN:=tmrPulseON.Q,PT:=T#0.5s);
IF tmrPulseON.Q THEN
	b500msPulse := TRUE;
ELSE
	b500msPulse := FALSE;
END_IF
pStation^.b500msPulse := b500msPulse;

(*Clear status fifo buffers*)
pStation^.AttentionRequiredFIFO.INIT(pFIFO:=ADR(pStation^.AttentionRequiredFIFOBuffer));
pStation^.NotOKtoStopFIFO.INIT(pFIFO:=ADR(pStation^.NotOKToStopFIFOBuffer));
pStation^.FaultedFIFO.INIT(pFIFO:=ADR(pStation^.FaultedFIFOBuffer));
pStation^.CycleManualFIFO.INIT(pFIFO:=ADR(pStation^.CycleManualFIFOBuffer));

(*Reset all manual bits*)
hiGateLock := 0;
hiGateUnlock :=0;

ACTION Input:
onsStart(CLK:=(pStation^.hiCycleStart OR Globals.iCycleStart));
cmdStart := onsStart.Q;
pStation^.hiCycleStart:=FALSE;

onsOperatorStop(CLK:=(pStation^.hiCycleStop OR Globals.iCycleStop));
cmdOperatorStop := onsOperatorStop.Q;
pStation^.hiCycleStop:=FALSE;

(*Machine stop receives signals from other stations or SCADA*)
onsMachineStop(CLK:=FALSE);
cmdMachineStop := pStation^.MachineStopRqst;
pStation^.MachineStopRqst := FALSE;

onsFaultAcknowledge(CLK:=(pStation^.hiFaultAck));
cmdFaultAcknowledge := onsFaultAcknowledge.Q;
pStation^.hiFaultAck:=FALSE;

onsFaultReset(CLK:=(pStation^.hiFaultReset));
cmdFaultReset :=onsFaultReset.Q;
pStation^.hiFaultReset:=FALSE;

onsStationReset(CLK:=(pStation^.hiStationReset));
cmdFullInit := onsStationReset.Q;
pStation^.hiStationReset:=FALSE;

onsSingleStepOn(CLK:=(pStation^.hiSingleStepON ));
cmdSingleStepOn := onsSingleStepOn.Q;
pStation^.hiSingleStepON:=FALSE;

onsSingleStepOff(CLK:=(pStation^.hiSingleStepOff ));
cmdSingleStepOff := onsSingleStepOff.Q;
pStation^.hiSingleStepOff:=FALSE;

onsSingleStepAdvance(CLK:=(pStation^.hiSingleStepAdvance ));
cmdSingleStepAdvance := onsSingleStepAdvance.Q;
pStation^.hiSingleStepAdvance:=FALSE;

onsManualMode(CLK:=(pStation^.hiManualMode ));
cmdManualMode := onsManualMode.Q;
pStation^.hiManualMode:=FALSE;
END_ACTION

END_PROGRAM

// ---- POUs/Stn100/Stn100_01_HMI.TcPOU
PROGRAM Stn100_01_HMI
VAR_IN_OUT
END_VAR
VAR
	pStation: POINTER TO Station;
	pStats: POINTER TO Component_Stats;

	State: DINT;
	NextState: DINT;
	FirstEntry: BOOL;
	tmrState: TON;
	tmrState20: TON;
	hoMessageTrigger: BOOL := FALSE;

	StationResetRequest: BOOL;
	hiStart: BOOL;
	hiStop: BOOL;
	hoStartButtonColor: DINT;
	hoStopButtonColor: DINT;
	ActiveMsg: HMIMessage;
	index: DINT;
	Msg: STRING;
	TimeStr: STRING;
	senMessageTriggerReset: FB_Sensor;
	hoMainBanner: HMIBanner;
	hiMessageReceived: BOOL :=FALSE;
	cColor: Colors;
END_VAR

pStation := ADR(Globals.gStation100);
pStats := ADR(Globals.gStn100_02_Stats);

IF pStation^.CycleAuto THEN
	hoStartButtonColor := cColor.Green;
	hoStopButtonColor := cColor.Grey;
ELSE
	hoStartButtonColor := cColor.Grey;
	hoStopButtonColor := cColor.Red;
END_IF

IF NextState <> State THEN
	(*code: Log state change into buffer*)
	FirstEntry := TRUE;
	State := NextState;
ELSE
	FirstEntry := FALSE;
END_IF

IF FirstEntry THEN
	tmrState(IN:=FALSE);
	tmrState20(IN:=FALSE);
END_IF

senMessageTriggerReset(Input := hoMessageTrigger, DelayON:=T#0.0S, DelayOFF:=T#1.0S);

CASE State OF

0:	(*Check FIFO for message. If msg, then unload*)
	IF pStation^.HMIMessageFIFO.Count  > 0 THEN
		pStation^.HMIMessageFIFO.REMOVE(pFIFO:=ADR(pStation^.HMIMessageBuffer), out=> ActiveMsg);
		(*If this is an empty message, don't pass it to the HMI*)
		IF ActiveMsg.Text <> '' AND ActiveMsg.Text <> ' ' THEN
			hoMessageTrigger := TRUE;
			NextState:=10;
		END_IF
	END_IF

10:	(*Wait for confirmation from HMI*)
	tmrState(IN:=TRUE, PT:=T#2.0S);
	IF hiMessageReceived OR tmrState.Q THEN
		hoMessageTrigger := FALSE;
		hiMessageReceived := FALSE;
		NextState:=20;
	END_IF
	IF  tmrState.Q THEN
		hiMessageReceived := FALSE;
		hoMessageTrigger := FALSE;
		NextState:=0;
	END_IF

20:	(*Clear*)
	tmrState20(IN:=TRUE, PT:=T#1.5S);
	IF NOT hiMessageReceived THEN
		NextState:=0;
	END_IF
	IF  tmrState20.Q THEN
		hiMessageReceived := FALSE;
		hoMessageTrigger := FALSE;
		NextState:=0;
	END_IF
END_CASE

(*Message banner*)
IF LEN(pStation^.FirstFault.StringData[0]) > 0 THEN
	hoMainBanner.Text :=pStation^.FirstFault.StringData[0];
	hoMainBanner.AltText :=pStation^.FirstFault.StringData[1];
	hoMainBanner.Color := cColor.Red;
ELSIF LEN(pStation^.OperatorMessage.Text) > 0 THEN
	hoMainBanner.Text :=pStation^.OperatorMessage.Text;
	hoMainBanner.AltText :=pStation^.OperatorMessage.AltText;
	hoMainBanner.Color := pStation^.OperatorMessage.Color;
ELSIF LEN(pStation^.StationMessage.Text) > 0 THEN
	hoMainBanner.Text :=pStation^.StationMessage.Text;
	hoMainBanner.AltText :=pStation^.StationMessage.AltText;
	hoMainBanner.Color := pStation^.StationMessage.Color;;
END_IF

END_PROGRAM

// ---- POUs/FB_Sensor.TcPOU
FUNCTION_BLOCK FB_Sensor
(*Sensor Debounce
ON is TRUE after Input has been TRUE for DelayON milliseconds
ON is FALSE after Input has been FALSE for DelayOFF milliseconds*)

VAR_INPUT
	Input: BOOL; (*Raw physical input*)
	DelayON: TIME; (*ON debounce time in milliseconds*)
	DelayOFF: TIME; (*OFF debounce time in milliseconds*)
END_VAR

VAR_OUTPUT
	ON: BOOL; (*Debounced input*)
END_VAR

VAR
	tmrDelayON: TON; (*Input ON debounce delay*)
	tmrDelayOFF: TON; (*Input OFF debounce delay*)
	InputON: R_TRIG; (*Rising edge Input ON debounced*)
	InputOFF: R_TRIG; (*Rising edge Input OFF debounced*)
END_VAR

(*Debounce timers*)
tmrDelayON(IN:=Input,PT:=DelayON);
tmrDelayOFF(IN:=NOT(Input),PT:=DelayOFF);

(*Rising edge of debounce timer outputs*)
InputON(CLK:=tmrDelayON.Q);
InputOFF(CLK:=tmrDelayOFF.Q);

(*Debounced Input Logic*)
IF InputON.Q THEN
	ON:=TRUE;
END_IF
IF InputOFF.Q THEN
	ON:=FALSE;
END_IF

END_FUNCTION_BLOCK

// ---- POUs/Stn100/Stn100_02_Stats.TcPOU
PROGRAM Stn100_02_Stats
VAR
	pStats: POINTER TO Component_Stats;
	pStation: POINTER TO Station;
	Local: FrameworkLocal;
	Framework: FB_Framework;

	tmrDelayStatsStart:TON;
	StartStats:R_TRIG;
	CurrentTime : TimeStamp;
	TimeStamp: StateTimeStamp;
	pStatsEventFifo : POINTER TO FIFO_StatsEvent;
	pStatsEventBuffer : POINTER TO StatsEventFIFOBuffer;
	ActiveEvent : StatsEvent;
	EventErrorCount : DINT;
	CurrentMode: DINT;
	NewMode : DINT;
	ModeStartTime: T_ULarge_Integer;
	TimeDiff : LREAL;
	CurrentFault : StatsFault;
	DbFaultRecord :StatsFault;
	CurrentFailure : StatsFailure;
	CurrentAggregate : StatsAggregateRecord;
	CurrentShiftAggregate : StatsShiftAggregateRecord;
	DBShiftOeeRecord :StatsShiftAggregateRecord;
	AggregateTimeCount : DINT;
	IntervalAggregateStart : R_TRIG;
	ShiftAggregateStart : R_TRIG;
	TempEvent : StatsEvent;
	LastMinute : DINT;
	idx : DINT;
	StartOfShift : BOOL;
	CurrentShiftIdx : DINT;
	TimeMins : DINT;
	MathTemp : DINT;
	CycleStartTime: LREAL;
	CycleStopTime: LREAL;
	CycleTimeBuffer : ARRAY [0..49] OF LREAL;
	CycleTimeIDX : DINT;
	CycleTimeAVG : LREAL;

	LastIdealCycleTime: LREAL := -1;
	TempIdealCycleTime: LREAL := -1;
	TempTotalParts: DINT;
	SumCycleTimeXParts: LREAL;
	onsIdealCycleTimeChange: R_TRIG;

	hoActiveShiftAggregate: StatsShiftAggregateRecord;
	hiActiveShiftIdx: DINT := 0;
	LastActiveShiftIndex: DINT := -1;
	nPeekCnt : DINT := 0;

	hoFaultLog : ARRAY[0..99] OF StatsFault;
	TempFaultRec : StatsFault;

	DB: FB_DBTransaction;
	DBTransact: udtDBTransact;
	StateFaultLogCheck : DINT;
	TempFaultRecord : StatsFault;
	spStoreFaultIn: udtDBStoreFault;
	spStoreFaultOut : udtDBStoreFault;
	DBFaultCount : DINT;
	tmrState20 : TON;
	tmrState40 : TON;
	tmrState60 : TON;
	tmrFaultTransCmp :TON;
	tmrFaultLogReset :TON;
	tmrFaultLogRetry :TON;
	ZeroTime :TIME;
	cTransaction: udtConstantsTransactions;
	cColor: Colors;
	cChannel: Channels;
END_VAR

IF Globals.gFirstScan THEN
	pStation := ADR(Globals.gStation100);
	pStats := ADR(Globals.gStn100_02_Stats);
	Local.pStateTraceBuffer := ADR(Globals.gStn100_StateTraceBuffer);
	Local.pStateTraceFifo := ADR(Globals.gStn100_StateTraceFifo);
	Local.FaultTimeLong := T#20000ms;
	Local.FaultTimeShort := T#10000ms;
	DefineMessages();
	DBTransact.pDatabaseInterface := ADR(Globals.gDatabaseInterface);
	DBTransact.UserID := pStation^.StationID * 100 + pStats^.Framework.ComponentIDRecord.ID;

	pStatsEventFifo := ADR(pStats^.StatsEventFIFO);
	pStatsEventBuffer := ADR(pStats^.StatsEventBuffer);
	pStats^.StatsEventFIFO.INIT(pFifo := ADR(pStats^.StatsEventBuffer));
	pStats^.StatsAggregateFIFO.INIT(pFifo := ADR(pStats^.StatsAggregateBuffer));
	MEMSET(ADR(CurrentAggregate),0,SIZEOF(CurrentAggregate));
	pStats^.StatsShiftAggregateFIFO.INIT(pFIFO := ADR(pStats^.StatsShiftAggregateBuffer));
	MEMSET(ADR(CurrentShiftAggregate),0,SIZEOF(CurrentShiftAggregate));
	pStats^.StatsFaultLog.INIT(pFIFO := ADR(pStats^.StatsFaultLogBuffer));
	pStats^.StatsFailureLog.INIT(pFIFO := ADR(pStats^.StatsFailureLogBuffer));
	LastIdealCycleTime := pStats^.IdealCycleTime;
	pStats^.StatsIdealCycleTimeFIFO.INIT(pFIFO := ADR(pStats^.StatsIdealCycleTimeBuffer));
	pStats^.StatsPartCountFIFO.INIT(pFIFO := ADR(pStats^.StatsPartCountBuffer));
	
	CycleTimeIDX := 0;
	hoActiveShiftAggregate := CurrentShiftAggregate;
	tmrFaultTransCmp(in:=FALSE,pt:=T#750MS);
	tmrFaultLogReset(in:=FALSE,pt:=T#10000MS);
	tmrFaultLogRetry(in:=FALSE,pt:=T#1000MS);	
END_IF

FrameWork(pFramework:=ADR(pStats^.Framework), pLocal:=ADR(Local), pStation:=pStation);
DB(pDBTransact:= ADR(DBTransact)); (*call transaction manager*)
CheckFaultLog();

CurrentTime := Globals.gCurrentTime;
tmrDelayStatsStart(in:=TRUE,pt:=t#50ms);
StartStats(clk:=tmrDelayStatsStart.q);
Globals.gCurrentHour := CurrentTime.DateTime.wHour;

IF StartStats.Q THEN
	ModeStartTime := CurrentTime.CurrentValue;
	LastMinute := CurrentTime.DateTime.wMinute;
	CurrentShiftAggregate.ShiftStartTimeStamp := CurrentTime;
	(*Determine what shift it is. 3rd shift is assumed to start before midnight*)
	TimeMins := CurrentTime.DateTime.wHour*60  + CurrentTime.DateTime.wMinute;
	MathTemp :=pStats^.StartOfShift[0,1] * 60 + pStats^.StartOfShift[0,0];
	IF (pStats^.StartOfShift[0,1] * 60 + pStats^.StartOfShift[0,0] - TimeMins) > 0 THEN
		CurrentShiftIdx := 2; (*3rd shift*)
	ELSIF  (pStats^.StartOfShift[1,1] * 60 + pStats^.StartOfShift[1,0] - TimeMins) > 0 THEN
		CurrentShiftIdx := 0; (*1st shift*)
	ELSIF  (pStats^.StartOfShift[2,1] * 60 + pStats^.StartOfShift[2,0] - TimeMins) > 0 THEN
		CurrentShiftIdx := 1; (*2nd shift*)
	ELSE
		CurrentShiftIdx := 2; (*3rd shift*)
	END_IF
	CurrentShiftAggregate.Shift := CurrentShiftIdx;
	CurrentShiftAggregate.ShiftStartTimeStamp := CurrentTime;
	Globals.gCurrShift :=CurrentShiftAggregate.Shift;

	(*On startup, it takes a few plc cycles to have a valid current time. Check to see if any events are already
	   in the buffer. If so, set their timestamp to the now valid current time.*)
	IF pStats^.StatsEventFIFO.Count  > 0 THEN
		FOR idx := 0 TO (pStats^.StatsEventFIFO.Count -1) DO
			pStats^.StatsEventBuffer.Buffer[idx].TimeStamp := CurrentTime;
	 	END_FOR
	END_IF
END_IF


IF (CurrentTime.DateTime.wMinute <> LastMinute) THEN
	(*Check for end of shift*)
	FOR idx := 0 TO 2 DO
		IF CurrentTime.DateTime.wHour  = pStats^.StartOfShift[idx,1] AND CurrentTime.DateTime.wMinute = pStats^.StartOfShift[idx,0] THEN
			StartOfShift := TRUE;
			CurrentShiftIdx := idx;
			MemCPY(ADR(DBShiftOeeRecord),ADR(CurrentShiftAggregate),SIZEOF(CurrentShiftAggregate));
			TempEvent.EType := Globals.cStats.Aggregate;
			TempEvent.Data[0] := DINT_TO_REAL(CurrentShiftIdx+1); (*Indicates to Aggregate to reset the CurrentShift data*)
			F_SendEvent(pStatsEventFifo, pStatsEventBuffer, ADR(TempEvent));
		END_IF
	END_FOR;

	(*Aggregate Interval*)
	IF (CurrentTime.DateTime.wMinute MOD pStats^.AggregateInterval ) = 0 AND NOT StartOfShift THEN
		TempEvent.EType := Globals.cStats.Aggregate;
		TempEvent.Data[0] := 0;
		F_SendEvent(pStatsEventFifo, pStatsEventBuffer, ADR(TempEvent));
	END_IF

	StartOfShift := FALSE;
	LastMinute :=CurrentTime.DateTime.wMinute;
	Globals.gCurrShift :=CurrentShiftAggregate.Shift;
END_IF

(*Ideal Cycle time changed*)
onsIdealCycleTimeChange(CLK:=(LastIdealCycleTime <> pStats^.IdealCycleTime));
IF onsIdealCycleTimeChange.Q THEN
	TempEvent.EType := Globals.cStats.Aggregate;
	TempEvent.Data[0] := 0;
	F_SendEvent(pStatsEventFifo, pStatsEventBuffer, ADR(TempEvent));
END_IF

(**********************
    Sequence logic
***********************)
CASE Local.State OF

0:	(*Wait for Start*)
	IF  Local.FirstEntry THEN
		;
	END_IF
	Local.OKToStop := TRUE;
	IF pStats^.StatsEventFIFO.Count  > 0 THEN
		pStats^.StatsEventFIFO.REMOVE(pFIFO:=pStatsEventBuffer, out=> ActiveEvent);
		IF  ActiveEvent.EType > 0 AND ActiveEvent.EType < 200 THEN
			(*Aggregate or Mode change*)
			Local.NextState := 100;
		ELSIF ActiveEvent.EType >=200 AND ActiveEvent.EType < 300 THEN
			(*Count only*)
			Local.NextState := 200;
		ELSIF ActiveEvent.EType >=300 AND ActiveEvent.EType < 400 THEN
			(*Process*)
			Local.NextState := 300;
		ELSE
			(*Error*)
			EventErrorCount := EventErrorCount + 1;
		END_IF
	END_IF

100:	(*Process mode change*)
	IF  Local.FirstEntry THEN
		TimeDiff := UINT64_TO_LREAL(UInt64Sub64(ActiveEvent.TimeStamp.CurrentValue,ModeStartTime)) / 600000000; (*time in minutes*)
		IF ActiveEvent.EType <> CurrentMode THEN
			(*do something*);
			CASE CurrentMode OF
				0 :	(*software startup*)
					NewMode := Globals.cStats.MachineStop;

				Globals.cStats.MachineStop :
					IF ActiveEvent.EType <> Globals.cStats.FaultAcknowledge AND	ActiveEvent.EType <> Globals.cStats.Faulted THEN
						(*mode change is valid*)
						CurrentAggregate.AutoStopTime := CurrentAggregate.AutoStopTime + TimeDiff;
						ModeStartTime := ActiveEvent.TimeStamp.CurrentValue;
						IF ActiveEvent.EType <> Globals.cStats.Aggregate THEN
							NewMode := ActiveEvent.EType;
						END_IF
					ELSE
						EventErrorCount := EventErrorCount + 1;
					END_IF

				Globals.cStats.OperatorStop :
					IF ActiveEvent.EType <> Globals.cStats.FaultAcknowledge AND	ActiveEvent.EType <> Globals.cStats.Faulted THEN
						(*mode change is valid*)
						CurrentAggregate.OperatorStopTime := CurrentAggregate.OperatorStopTime + TimeDiff;
						ModeStartTime := ActiveEvent.TimeStamp.CurrentValue;
						IF ActiveEvent.EType <> Globals.cStats.Aggregate THEN
							NewMode := ActiveEvent.EType;
						END_IF
					ELSE
						EventErrorCount := EventErrorCount + 1;
					END_IF

				Globals.cStats.Working :
					IF ActiveEvent.EType <> Globals.cStats.FaultAcknowledge   THEN
						(*mode change is valid*)
						CurrentAggregate.WorkTime := CurrentAggregate.WorkTime + TimeDiff;
						ModeStartTime := ActiveEvent.TimeStamp.CurrentValue;
						IF ActiveEvent.EType <> Globals.cStats.Aggregate THEN
							NewMode := ActiveEvent.EType;
						END_IF
					ELSE
						EventErrorCount := EventErrorCount + 1;
					END_IF

				Globals.cStats.Bypass :
					IF ActiveEvent.EType <> Globals.cStats.FaultAcknowledge   THEN
						(*mode change is valid*)
						CurrentAggregate.BypassTime := CurrentAggregate.BypassTime + TimeDiff;
						ModeStartTime := ActiveEvent.TimeStamp.CurrentValue;
						IF ActiveEvent.EType <> Globals.cStats.Aggregate THEN
							NewMode := ActiveEvent.EType;
						END_IF
					ELSE
						EventErrorCount := EventErrorCount + 1;
					END_IF

				Globals.cStats.Blocked :
					IF ActiveEvent.EType <> Globals.cStats.FaultAcknowledge   THEN
						(*mode change is valid*)
						CurrentAggregate.BlockTime := CurrentAggregate.BlockTime + TimeDiff;
						ModeStartTime := ActiveEvent.TimeStamp.CurrentValue;
						IF ActiveEvent.EType <> Globals.cStats.Aggregate THEN
							NewMode := ActiveEvent.EType;
						END_IF
					ELSE
						EventErrorCount := EventErrorCount + 1;
					END_IF

				Globals.cStats.Starved :
					IF ActiveEvent.EType <> Globals.cStats.FaultAcknowledge   THEN
						(*mode change is valid*)
						CurrentAggregate.StarveTime := CurrentAggregate.StarveTime + TimeDiff;
						ModeStartTime := ActiveEvent.TimeStamp.CurrentValue;
						IF ActiveEvent.EType <> Globals.cStats.Aggregate THEN
							NewMode := ActiveEvent.EType;
						END_IF
					ELSE
						EventErrorCount := EventErrorCount + 1;
					END_IF

				Globals.cStats.Empty :
					IF ActiveEvent.EType <> Globals.cStats.FaultAcknowledge   THEN
						(*mode change is valid*)
						CurrentAggregate.EmptyTime := CurrentAggregate.EmptyTime + TimeDiff;
						ModeStartTime := ActiveEvent.TimeStamp.CurrentValue;
						IF ActiveEvent.EType <> Globals.cStats.Aggregate THEN
							NewMode := ActiveEvent.EType;
						END_IF
					ELSE
						EventErrorCount := EventErrorCount + 1;
					END_IF

				Globals.cStats.Retry :
					IF ActiveEvent.EType <> Globals.cStats.FaultAcknowledge   THEN
						(*mode change is valid*)
						CurrentAggregate.EmptyTime := CurrentAggregate.EmptyTime + TimeDiff;
						ModeStartTime := ActiveEvent.TimeStamp.CurrentValue;
						IF ActiveEvent.EType <> Globals.cStats.Aggregate THEN
							NewMode := ActiveEvent.EType;
						END_IF
					ELSE
						EventErrorCount := EventErrorCount + 1;
					END_IF

				Globals.cStats.Mastering :
					IF ActiveEvent.EType <> Globals.cStats.FaultAcknowledge   THEN
						(*mode change is valid*)
						CurrentAggregate.MasterTime := CurrentAggregate.MasterTime + TimeDiff;
						ModeStartTime := ActiveEvent.TimeStamp.CurrentValue;
						IF ActiveEvent.EType <> Globals.cStats.Aggregate THEN
							NewMode := ActiveEvent.EType;
						END_IF
					ELSE
						EventErrorCount := EventErrorCount + 1;
					END_IF

				Globals.cStats.Faulted :
					IF ActiveEvent.EType <> Globals.cStats.OperatorStop OR ActiveEvent.EType <> Globals.cStats.MachineStop   THEN
						(*mode change is valid*)
						IF ActiveEvent.EType = Globals.cStats.FaultAcknowledge THEN
							CurrentFault.AcknowledgeTime := TimeDiff;
						ELSE
							CurrentAggregate.FaultTime := CurrentAggregate.FaultTime + TimeDiff;
							ModeStartTime := ActiveEvent.TimeStamp.CurrentValue;
							IF ActiveEvent.EType <> Globals.cStats.Aggregate THEN
								CurrentFault.Duration := UINT64_TO_LREAL(UInt64Sub64( ActiveEvent.TimeStamp.CurrentValue,CurrentFault.TimeStamp.CurrentValue)) / 600000000;
								IF CurrentFault.AcknowledgeTime = 0 THEN
									CurrentFault.AcknowledgeTime := CurrentFault.Duration;
									EventErrorCount := EventErrorCount + 1;
								END_IF
								NewMode := ActiveEvent.EType;
								pStats^.StatsFaultLog.INSERT(pFIFO:=ADR(pStats^.StatsFaultLogBuffer), in:=CurrentFault);
							END_IF
						END_IF
					ELSE
						EventErrorCount := EventErrorCount + 1;
					END_IF
			END_CASE

			IF NewMode <> CurrentMode THEN
				(*need to handle new event specifics*)
				CASE NewMode OF
					Globals.cStats.MachineStop :
						CurrentAggregate.AutoStopCount := CurrentAggregate.AutoStopCount + 1;
					Globals.cStats.OperatorStop :
						CurrentAggregate.OperatorStopCount := CurrentAggregate.OperatorStopCount + 1;
					Globals.cStats.Working :
						CurrentAggregate.WorkCount := CurrentAggregate.WorkCount + 1;
					Globals.cStats.Bypass :
						CurrentAggregate.BypassCount := CurrentAggregate.BypassCount + 1;
					Globals.cStats.Blocked :
						CurrentAggregate.BlockCount := CurrentAggregate.BlockCount + 1;
					Globals.cStats.Starved :
						CurrentAggregate.StarveCount := CurrentAggregate.StarveCount + 1;
					Globals.cStats.Empty :
						CurrentAggregate.EmptyCount := CurrentAggregate.EmptyCount + 1;
					Globals.cStats.Retry :
						CurrentAggregate.RetryCount := CurrentAggregate.RetryCount + 1;
					Globals.cStats.Mastering :
						CurrentAggregate.MasterCount := CurrentAggregate.MasterCount + 1;
					Globals.cStats.Faulted :
						CurrentAggregate.FaultCount := CurrentAggregate.FaultCount + 1;
						MEMSET(ADR(CurrentFault),0,SIZEOF(CurrentFault));
						CurrentFault.TimeStamp := ActiveEvent.TimeStamp;
						CurrentFault.FaultID := REAL_TO_DINT(ActiveEvent.Data[0]);
						CurrentFault.StationID := pStation^.StationID;
						CurrentFault.Data[0] := ActiveEvent.Data[1];
						CurrentFault.Data[1] := ActiveEvent.Data[2];
						CurrentFault.Data[2] := ActiveEvent.Data[3];
						CurrentFault.StringData := ActiveEvent.StringData;
		
					ELSE
						EventErrorCount := EventErrorCount + 1;
				END_CASE
				CurrentMode:=NewMode;
			END_IF
			IF ActiveEvent.EType = Globals.cStats.Aggregate THEN
				Aggregate();
			END_IF
		END_IF
	END_IF
	Local.NextState := 0;

200:	(*Count only events*)
	CASE ActiveEvent.EType OF
		Globals.cStats.Failure :
			CurrentAggregate.RejectCount := CurrentAggregate.RejectCount + REAL_TO_INT(ActiveEvent.Data[1]);
			CurrentFailure.TimeStamp := ActiveEvent.TimeStamp;
			CurrentFailure.StationID := pStation^.StationID;
			CurrentFailure.FailureID := REAL_TO_INT(ActiveEvent.Data[0]);
			CurrentFailure.Parameters := ActiveEvent.StringData[0];
			Globals.gShiftData[Globals.gCurrShift].ScrapCount := CurrentAggregate.RejectCount;
			Globals.gHourlyData[Globals.gCurrentHour].ScrapCount := CurrentAggregate.RejectCount;
			pStats^.StatsFailureLog.INSERT(pFIFO:=ADR(pStats^.StatsFailureLogBuffer), in:=CurrentFailure);
		Globals.cStats.Good :
			CurrentAggregate.GoodCount := CurrentAggregate.GoodCount + REAL_TO_INT(ActiveEvent.Data[0]);
			Globals.gShiftData[Globals.gCurrShift].GoodCount := Globals.gShiftData[Globals.gCurrShift].GoodCount + REAL_TO_INT(ActiveEvent.Data[0]);
			Globals.gHourlyData[Globals.gCurrentHour].GoodCount := Globals.gHourlyData[Globals.gCurrentHour].GoodCount + REAL_TO_INT(ActiveEvent.Data[0]);		
		Globals.cStats.FirstTimeGood :
			CurrentAggregate.FirstTimeGoodCount := CurrentAggregate.FirstTimeGoodCount + 1;
		Globals.cStats.FirstTimeStart :
			CurrentAggregate.FirstTimeStartCount := CurrentAggregate.FirstTimeStartCount + 1;
		Globals.cStats.Initialize :
			CurrentAggregate.InitCount := CurrentAggregate.InitCount + 1;
		ELSE
			EventErrorCount := EventErrorCount + 1;
	END_CASE;
	Local.NextState := 0;

300:	(*Process data events *)
	IF  Local.FirstEntry THEN
	CASE ActiveEvent.EType OF
		Globals.cStats.CycleTime :
			CASE REAL_TO_INT(ActiveEvent.Data[0]) OF
				0: (*Start timer*)
					CycleStartTime := UINT64_TO_LREAL( ActiveEvent.TimeStamp.CurrentValue);
				1: (*Cancel timer*)
					CycleStartTime :=0;
				2: (*End of good cycle time*)
					IF CycleStartTime > 0 THEN
						CycleStopTime := UINT64_TO_LREAL( ActiveEvent.TimeStamp.CurrentValue);
						IF CycleTimeIDX >= 50 THEN (* Start overwriting oldest elements *)
							CycleTimeIDX := 0;
						END_IF
						CycleTimeBuffer[CycleTimeIDX] := (CycleStopTime - CycleStartTime ) / 10000000; (*cycle time is in seconds*)
						CycleTimeIDX := CycleTimeIDX + 1;
					END_IF
				ELSE
					EventErrorCount := EventErrorCount + 1;
			END_CASE;
		ELSE
			EventErrorCount := EventErrorCount + 1;
	END_CASE;
		Local.NextState := 0;
	END_IF

5000 :
	Local.NextState := 0;

END_CASE

(*0 is current, 1 is 1st most recent FIFO *)
IF(hiActiveShiftIdx <> LastActiveShiftIndex) THEN
	LastActiveShiftIndex := hiActiveShiftIdx;
	IF (hiActiveShiftIdx > 0) AND (hiActiveShiftIdx <=270) THEN
		IF hiActiveShiftIdx > pStats^.StatsShiftAggregateFIFO.Count THEN
			hiActiveShiftIdx := pStats^.StatsShiftAggregateFIFO.Count;
		END_IF
	
		nPeekCnt := pStats^.StatsShiftAggregateFIFO.Count - hiActiveShiftIdx;
		pStats^.StatsShiftAggregateFIFO.PEEK(pFIFO:=ADR(pStats^.StatsShiftAggregateBuffer), PeekCnt := nPeekCnt, out=> hoActiveShiftAggregate);
	
	ELSE
		hoActiveShiftAggregate := CurrentShiftAggregate;
	END_IF
END_IF
(**********************
  END of Sequence logic
***********************)

ACTION Aggregate:
(*Average cycle TIME*)
IF CycleTimeIDX > 0 THEN
	CycleTimeAVG := 0;
	FOR idx := 0 TO (CycleTimeIDX-1) DO
		CycleTimeAVG := CycleTimeAVG + CycleTimeBuffer[idx];
	END_FOR;
	CycleTimeAVG := CycleTimeAVG / idx;
	CurrentAggregate.GoodCycleTime := CycleTimeAVG;


	CurrentShiftAggregate.CycleTimeAvgSum := CurrentShiftAggregate.CycleTimeAvgSum + CycleTimeAVG;
	CurrentShiftAggregate.CycleTimeAvgCnt := CurrentShiftAggregate.CycleTimeAvgCnt + 1;

	IF CurrentShiftAggregate.CycleTimeAvgCnt <> 0 THEN
		CurrentShiftAggregate.AggregateData.GoodCycleTime := CurrentShiftAggregate.CycleTimeAvgSum / CurrentShiftAggregate.CycleTimeAvgCnt;
	END_IF

	CycleTimeIDX := 0;
END_IF

(*Aggregate data*)
CurrentShiftAggregate.AggregateData.Shift := CurrentShiftAggregate.Shift;
CurrentShiftAggregate.AggregateData.AutoStopCount := CurrentShiftAggregate.AggregateData.AutoStopCount + CurrentAggregate.AutoStopCount;
CurrentShiftAggregate.AggregateData.AutoStopTime :=CurrentShiftAggregate.AggregateData.AutoStopTime+CurrentAggregate.AutoStopTime;
CurrentShiftAggregate.AggregateData.BlockCount :=CurrentShiftAggregate.AggregateData.BlockCount+CurrentAggregate.BlockCount;
CurrentShiftAggregate.AggregateData.BlockTime :=CurrentShiftAggregate.AggregateData.BlockTime+CurrentAggregate.BlockTime;
CurrentShiftAggregate.AggregateData.BypassCount :=CurrentShiftAggregate.AggregateData.BypassCount+CurrentAggregate.BypassCount;
CurrentShiftAggregate.AggregateData.BypassTime :=CurrentShiftAggregate.AggregateData.BypassTime+CurrentAggregate.BypassTime;
CurrentShiftAggregate.AggregateData.EmptyCount :=CurrentShiftAggregate.AggregateData.EmptyCount+CurrentAggregate.EmptyCount;
CurrentShiftAggregate.AggregateData.EmptyTime :=CurrentShiftAggregate.AggregateData.EmptyTime+CurrentAggregate.EmptyTime;
CurrentShiftAggregate.AggregateData.FaultCount :=CurrentShiftAggregate.AggregateData.FaultCount +CurrentAggregate.FaultCount;
CurrentShiftAggregate.AggregateData.FaultTime :=CurrentShiftAggregate.AggregateData.FaultTime+CurrentAggregate.FaultTime;
CurrentShiftAggregate.AggregateData.FirstTimeGoodCount :=CurrentShiftAggregate.AggregateData.FirstTimeGoodCount+CurrentAggregate.FirstTimeGoodCount;
CurrentShiftAggregate.AggregateData.FirstTimeStartCount :=CurrentShiftAggregate.AggregateData.FirstTimeStartCount+CurrentAggregate.FirstTimeStartCount;
CurrentShiftAggregate.AggregateData.GoodCount :=CurrentShiftAggregate.AggregateData.GoodCount +CurrentAggregate.GoodCount;
CurrentShiftAggregate.AggregateData.InitCount :=CurrentShiftAggregate.AggregateData.InitCount+CurrentAggregate.InitCount;
CurrentShiftAggregate.AggregateData.MasterCount :=CurrentShiftAggregate.AggregateData.MasterCount +CurrentAggregate.MasterCount;
CurrentShiftAggregate.AggregateData.MasterTime :=CurrentShiftAggregate.AggregateData.MasterTime+CurrentAggregate.MasterTime;
CurrentShiftAggregate.AggregateData.OperatorStopCount :=CurrentShiftAggregate.AggregateData.OperatorStopCount+CurrentAggregate.OperatorStopCount;
CurrentShiftAggregate.AggregateData.OperatorStopTime :=CurrentShiftAggregate.AggregateData.OperatorStopTime+CurrentAggregate.OperatorStopTime;
CurrentShiftAggregate.AggregateData.OtherCount :=CurrentShiftAggregate.AggregateData.OtherCount +CurrentAggregate.OtherCount;
CurrentShiftAggregate.AggregateData.OtherTime :=CurrentShiftAggregate.AggregateData.OtherTime+CurrentAggregate.OtherTime;
CurrentShiftAggregate.AggregateData.RejectCount :=CurrentShiftAggregate.AggregateData.RejectCount +CurrentAggregate.RejectCount;
CurrentShiftAggregate.AggregateData.RetryCount :=CurrentShiftAggregate.AggregateData.RetryCount+CurrentAggregate.RetryCount;
CurrentShiftAggregate.AggregateData.RetryTime :=CurrentShiftAggregate.AggregateData.RetryTime +CurrentAggregate.RetryTime;
CurrentShiftAggregate.AggregateData.StarveCount :=CurrentShiftAggregate.AggregateData.StarveCount +CurrentAggregate.StarveCount;
CurrentShiftAggregate.AggregateData.StarveTime :=CurrentShiftAggregate.AggregateData.StarveTime +CurrentAggregate.StarveTime;
CurrentShiftAggregate.AggregateData.WorkCount :=CurrentShiftAggregate.AggregateData.WorkCount+CurrentAggregate.WorkCount;
CurrentShiftAggregate.AggregateData.WorkTime :=CurrentShiftAggregate.AggregateData.WorkTime +CurrentAggregate.WorkTime;

(*OEE calculations*)

(*Available time*)
CurrentShiftAggregate.AvailableTime := UINT64_TO_LREAL(UInt64Sub64(ActiveEvent.TimeStamp.CurrentValue,
													CurrentShiftAggregate.ShiftStartTimeStamp.CurrentValue)) / 600000000;

(*Total down time*)
CurrentShiftAggregate.TotalDownTime := 	CurrentShiftAggregate.AggregateData.AutoStopTime +
									CurrentShiftAggregate.AggregateData.FaultTime +
									CurrentShiftAggregate.AggregateData.OperatorStopTime;

(*Planned down time*)
IF CurrentShiftAggregate.TotalDownTime  > pStats^.PlannedDowntime[CurrentShiftIdx] THEN
	CurrentShiftAggregate.PlannedDownTime :=pStats^.PlannedDowntime[CurrentShiftIdx];
ELSE
	CurrentShiftAggregate.PlannedDownTime :=CurrentShiftAggregate.TotalDownTime;
END_IF

(*Unplaned down time*)
CurrentShiftAggregate.UnplannedDownTime := CurrentShiftAggregate.TotalDownTime  - CurrentShiftAggregate.PlannedDownTime;
(*Net available time*)
CurrentShiftAggregate.NetAvailableTime := CurrentShiftAggregate.AvailableTime - CurrentShiftAggregate.PlannedDownTime;
(*Operating time*)
CurrentShiftAggregate.OperatingTime := CurrentShiftAggregate.NetAvailableTime - CurrentShiftAggregate.UnplannedDownTime;
(*Equipment availability*)
IF CurrentShiftAggregate.NetAvailableTime > 0 THEN
	CurrentShiftAggregate.EquipmentAvailability := CurrentShiftAggregate.OperatingTime  / CurrentShiftAggregate.NetAvailableTime * 100;
ELSE
	CurrentShiftAggregate.EquipmentAvailability := 0;
END_IF
(*Total parts*)
CurrentShiftAggregate.TotalParts := CurrentShiftAggregate.AggregateData.GoodCount + CurrentShiftAggregate.AggregateData.RejectCount;

(*Performance efficiency*)
(* Since Ideal Cycle time can change, keep track off all of the cycle times and the Total Parts for those cycle times *)
CurrentShiftAggregate.AggregateData.PartsForCurrentCycleTime :=
	CurrentShiftAggregate.AggregateData.PartsForCurrentCycleTime + CurrentAggregate.GoodCount + CurrentAggregate.RejectCount;

IF pStats^.IdealCycleTime <> LastIdealCycleTime THEN
	pStats^.StatsIdealCycleTimeFIFO.INSERT(pFIFO := ADR(pStats^.StatsIdealCycleTimeBuffer), in:=LastIdealCycleTime);
	pStats^.StatsPartCountFIFO.INSERT(pFIFO := ADR(pStats^.StatsPartCountBuffer), in:=CurrentShiftAggregate.AggregateData.PartsForCurrentCycleTime);

	LastIdealCycleTime := pStats^.IdealCycleTime;
	CurrentShiftAggregate.AggregateData.PartsForCurrentCycleTime := 0;
END_IF

IF CurrentShiftAggregate.OperatingTime > 0 THEN
	SumCycleTimeXParts :=
		pStats^.IdealCycleTime * CurrentShiftAggregate.AggregateData.PartsForCurrentCycleTime;

	FOR idx := 0 TO pStats^.StatsIdealCycleTimeFIFO.Count - 1 DO
		TempIdealCycleTime := pStats^.StatsIdealCycleTimeBuffer.Buffer[idx];
		TempTotalParts := pStats^.StatsPartCountBuffer.Buffer[idx];
		SumCycleTimeXParts := SumCycleTimeXParts + (TempIdealCycleTime * TempTotalParts);
	END_FOR
	(*CurrentShiftAggregate.PerformanceEfficiency := SumCycleTimeXParts / (CurrentShiftAggregate.OperatingTime * 60) * 100;*)

	CurrentShiftAggregate.PerformanceEfficiency := (pStats^.IdealCycleTime * CurrentShiftAggregate.TotalParts) / (CurrentShiftAggregate.OperatingTime * 60) * 100;
ELSE
	CurrentShiftAggregate.PerformanceEfficiency := 0;
END_IF


(*Quality rate*)
IF CurrentShiftAggregate.TotalParts > 0 THEN
	CurrentShiftAggregate.QualityRate := DINT_TO_REAL(CurrentShiftAggregate.AggregateData.GoodCount) / DINT_TO_REAL(CurrentShiftAggregate.TotalParts) * 100;
ELSE
	CurrentShiftAggregate.QualityRate := 0;
END_IF
(*OEE*)
CurrentShiftAggregate.OverallEquipmentEffectiveness := CurrentShiftAggregate.EquipmentAvailability *
												CurrentShiftAggregate.QualityRate *
												CurrentShiftAggregate.PerformanceEfficiency * 0.0001;

(*Insert current aggregate into aggregate log*)
CurrentAggregate.TimeStamp := ActiveEvent.TimeStamp;
CurrentAggregate.Shift := CurrentShiftAggregate.Shift;
pStats^.StatsAggregateFIFO.INSERT(pFIFO := ADR(pStats^.StatsAggregateBuffer), in:=CurrentAggregate);
MEMSET(ADR(CurrentAggregate),0,SIZEOF(CurrentAggregate));

(* Ensure Active shift gets updatad on HMI *)
LastActiveShiftIndex := -1;

(*check for end of shift*)
IF REAL_TO_INT(ActiveEvent.Data[0]) > 0 THEN
	CurrentShiftAggregate.AggregateData.TimeStamp := ActiveEvent.TimeStamp;
	pStats^.StatsShiftAggregateFIFO.INSERT(pFIFO := ADR(pStats^.StatsShiftAggregateBuffer), in:=CurrentShiftAggregate);
	MEMSET(ADR(CurrentShiftAggregate),0,SIZEOF(CurrentShiftAggregate));
	CurrentShiftAggregate.ShiftStartTimeStamp := ActiveEvent.TimeStamp;
	CurrentShiftAggregate.Shift := REAL_TO_DINT(ActiveEvent.Data[0] - 1);

	pStats^.StatsIdealCycleTimeFIFO.INIT(pFIFO := ADR(pStats^.StatsIdealCycleTimeBuffer));
	pStats^.StatsPartCountFIFO.INIT(pFIFO := ADR(pStats^.StatsPartCountBuffer));
	LastIdealCycleTime := pStats^.IdealCycleTime;

END_IF
END_ACTION

ACTION CheckFaultLog:
(**********************
 Check fault log for records. If found, send to database  
***********************)

tmrState20(IN:=StateFaultLogCheck = 20,PT:=T#10s);
tmrState40(IN:=StateFaultLogCheck = 30,PT:=T#10s);
tmrState60(IN:=StateFaultLogCheck = 60,PT:=T#10s);
CASE StateFaultLogCheck OF

0: 	(*Check fault log fifo*)

	IF pStats^.StatsFaultLog.Count > 0 THEN
		pStats^.StatsFaultLog.PEEK (pFIFO:=ADR(pStats^.StatsFaultLogBuffer), out=> TempFaultRecord);
		StateFaultLogCheck := 10;
	END_IF

10:	(*Call uspStoreFault*)

	spStoreFaultIn.Station := pStation^.StationID;
	spStoreFaultIn.FaultCode := TempFaultRecord.FaultID;
	spStoreFaultIn.FaultText := TempFaultRecord.StringData[0];
	spStoreFaultIn.AcknowledgeTime := TempFaultRecord.AcknowledgeTime;
	spStoreFaultIn.Duration := TempFaultRecord.Duration;
	spStoreFaultIn.TimeStamp.CurrentValue := TempFaultRecord.TimeStamp.CurrentValue;
	spStoreFaultIn.Data1 := TempFaultRecord.Data[0];
	spStoreFaultIn.Data2 := TempFaultRecord.Data[1];
	spStoreFaultIn.Data3 := TempFaultRecord.Data[2];
	spStoreFaultIn.StringData1 := TempFaultRecord.StringData[1];
	spStoreFaultIn.StringData2 := TempFaultRecord.StringData[2];
(*Copy the spStoreFaultIn data to the dbFaultRecord *)
	DbFaultRecord.TimeStamp := TempFaultRecord.TimeStamp;
	DbFaultRecord.FaultID := TempFaultRecord.FaultID;
	DbFaultRecord.StationID := pStation^.StationID;
	DbFaultRecord.Data[0] := TempFaultRecord.Data[0];
	DbFaultRecord.Data[1] := TempFaultRecord.Data[1];
	DbFaultRecord.Data[2] := TempFaultRecord.Data[2];
	DbFaultRecord.StringData := TempFaultRecord.StringData;
	DbFaultRecord.AcknowledgeTime := TempFaultRecord.AcknowledgeTime;
	DbFaultrecord.Duration := TempFaultRecord.Duration;
	MEMCPY(ADR(DBTransact.DataIn[0]),ADR(spStoreFaultIn),SIZEOF(spStoreFaultIn));
	DBTransact.DataLength := SIZEOF(spStoreFaultIn);
	DBTransact.TransactionID := cTransaction.StoreFault;
	DBTransact.Start := TRUE;
	StateFaultLogCheck := 20;
	Globals.gDbTransact[0].FaultedTranReq :=TRUE;

20:	(*Wait for done*)

	IF DBTransact.Done OR Globals.gDbTransact[0].FaultedTranCmp THEN
		StateFaultLogCheck := 30;
		DBTransact.Start := FALSE;
	END_IF
	IF tmrState20.Q THEN
		StateFaultLogCheck := 60;
		DBTransact.Start := FALSE;
		DBFaultCount := DBFaultCount + 1;
	END_IF

30: (*Get DB result*)
	MEMCPY(ADR(spStoreFaultOut),ADR(DBTransact.DataOut[0]),SIZEOF(spStoreFaultOut));
	IF spStoreFaultOut.ResultCode = 1  OR  Globals.gDbTransact[0].FaultedTranCmp THEN
		StateFaultLogCheck := 40;
	ELSE
		Local.MsgText := 'Stored Procedure error, ';
		Local.MsgText := CONCAT(Local.MsgText, DINT_TO_STRING(spStoreFaultOut.ResultCode));
		Local.MsgText := CONCAT(Local.MsgText, ': ');
		Local.MsgText := CONCAT(Local.MsgText, spStoreFaultOut.ResultText);
		Local.AltMsgText := 'No Alternate text';
		F_AddMessage(pStation, Local.MsgText, Local.AltMsgText, cColor.Red, cChannel.Fault);
		StateFaultLogCheck := 60;
		DBFaultCount := DBFaultCount + 1;
	END_IF

40:

	IF NOT DBTransact.Done OR (Globals.gDbTransact[0].FaultedTranReq AND Globals.gDbTransact[0].FaultedTranCmp) THEN
		StateFaultLogCheck := 50;
	END_IF
	IF tmrState40.Q THEN
		StateFaultLogCheck := 60;
		DBFaultCount := DBFaultCount + 1;
	END_IF

50:
	Globals.gDbTransact[0].FaultedTranReq := FALSE;
	Globals.gDbTransact[0].FaultedTranCmp := FALSE;
	pStats^.StatsFaultLog.REMOVE(pFIFO:=ADR(pStats^.StatsFaultLogBuffer), out=> TempFaultRecord);
	StateFaultLogCheck := 0;

60:	(*Fault*)

	IF DBFaultCount < 3 THEN
		IF tmrState60.Q THEN
			StateFaultLogCheck := 10;
		END_IF
	ELSE
		DBFaultCount := 0;
		StateFaultLogCheck := 50;
	END_IF

END_CASE
END_ACTION

ACTION DefineMessages:
(*Define your Message Structure Here*)
Local.MsgArray[0].Id := 1;
Local.MsgArray[0].Text := 'FaultMessage';
END_ACTION

END_PROGRAM

// ---- POUs/FB_DBTransaction.TcPOU
FUNCTION_BLOCK FB_DBTransaction

VAR_INPUT
	pDBTransact: POINTER TO udtDBTransact;
END_VAR

VAR_OUTPUT
	ErrorCode: DINT;
	ErrorMessage : STRING[256];
END_VAR

VAR
	NextState: DINT;
	FirstEntry: BOOL;
	tmrState: TON;
	idx: DINT;
	ChannelNum:SINT;
	TriggerMask:DWORD;

	Time1: TimeStamp;
	Time2: TimeStamp;
	Time3: TimeStamp;
	Time4: TimeStamp;

	StateTraceBuffer : TraceFIFOBuffer;
	StateTraceFifo : FIFO_StateTrace := ( Overwrite := TRUE );
	StateTimeStamp : StateTimeStamp;
	pStateTraceBuffer: POINTER TO TraceFIFOBuffer;

	Temp: DINT;
END_VAR

pStateTraceBuffer := ADR(StateTraceBuffer);

IF FirstEntry THEN
	tmrState(IN:=FALSE);
END_IF

IF pDBTransact^.UserID = 2 THEN
	Temp := pDBTransact^.UserID;
END_IF


CASE pDBTransact^.State OF

0:	(*Idle*)
	IF pDBTransact^.Start THEN
		pDBTransact^.State := 10;
		ErrorCode := 0;
		ErrorMessage :='';
		Time1:=F_GetTimeStamp();
	END_IF

10:
	FOR idx := 0 TO 19 DO
		IF pDBTransact^.pDatabaseInterface^.Connection[idx].CurrentUser = 0 OR
				pDBTransact^.pDatabaseInterface^.Connection[idx].CurrentUser = pDBTransact^.UserID THEN
			pDBTransact^.pDatabaseInterface^.Connection[idx].CurrentUser := pDBTransact^.UserID;
			ChannelNum := DINT_TO_SINT(idx);
			TriggerMask := REAL_TO_DWORD(EXPT(2,ChannelNum));
			pDBTransact^.State := 20;
			EXIT;
		END_IF
	END_FOR
	Time2:=F_GetTimeStamp();

20: (*Trigger Database*)
	MEMSET(ADR(pDBTransact^.DataOUT[0]),0,SIZEOF(pDBTransact^.DataOut));
	MEMCPY(ADR(pDBTransact^.pDatabaseInterface^.Connection[ChannelNum].DataIn[0]),
			ADR(pDBTransact^.TransactionID),
			SIZEOF(pDBTransact^.TransactionID));
	MEMCPY(ADR(pDBTransact^.pDatabaseInterface^.Connection[ChannelNum].DataIn[0+SIZEOF(pDBTransact^.TransactionID)]),
			ADR(pDBTransact^.DataIn[0]),
			pDBTransact^.DataLength);
	pDBTransact^.pDatabaseInterface^.Trigger := SETBIT32(pDBTransact^.pDatabaseInterface^.Trigger ,ChannelNum);
	Time3:=F_GetTimeStamp();
	pDBTransact^.State := 25;

25:
	IF (pDBTransact^.pDatabaseInterface^.Response AND TriggerMask) > 0 THEN
		MEMCPY(ADR(pDBTransact^.DataOUT[0]),
				ADR(pDBTransact^.pDatabaseInterface^.Connection[ChannelNum].DataOut[0+SIZEOF(pDBTransact^.TransactionID)]),
				pDBTransact^.DataLength);
		ErrorCode :=pDBTransact^.pDatabaseInterface^.Connection[ChannelNum].ErrorCode;
		ErrorMessage :=pDBTransact^.pDatabaseInterface^.Connection[ChannelNum].ErrorMessage;
		pDBTransact^.pDatabaseInterface^.Trigger :=CLEARBIT32(pDBTransact^.pDatabaseInterface^.Trigger,ChannelNum);
		pDBTransact^.State := 30;
	END_IF
	IF NOT pDBTransact^.Start THEN
		pDBTransact^.State := 40; (*if fault for timeout, need way out of state 25*)
		pDBTransact^.pDatabaseInterface^.Trigger :=CLEARBIT32(pDBTransact^.pDatabaseInterface^.Trigger,ChannelNum);
	END_IF

30:
	IF (pDBTransact^.pDatabaseInterface^.Response AND TriggerMask) = 0 THEN
		pDBTransact^.Done := TRUE;
		pDBTransact^.ErrorCode := ErrorCode;
		pDBTransact^.ErrorMessage := ErrorMessage;
		pDBTransact^.State := 40;
		Time4:=F_GetTimeStamp();
	END_IF

40:
	IF NOT pDBTransact^.Start THEN
		pDBTransact^.Done := FALSE;
		pDBTransact^.pDatabaseInterface^.Connection[ChannelNum].CurrentUser := 0;
		MEMSET(ADR(pDBTransact^.pDatabaseInterface^.Connection[ChannelNum].DataOut[0]),0,SIZEOF(pDBTransact^.pDatabaseInterface^.Connection[ChannelNum].DataOut));
		pDBTransact^.State := 0;
	END_IF

END_CASE

IF NextState <> pDBTransact^.state THEN
	FirstEntry := TRUE;
	NextState:= pDBTransact^.State;
	Time1 := F_GetTimeStamp();
	StateTimeStamp.ID := ChannelNum;
	StateTimeStamp.State := pDBTransact^.State;
	StateTimeStamp.TimeHi := Time1.CurrentValue.dwHighPart;
	StateTimeStamp.TimeLo:= Time1.CurrentValue.dwLowPart;
	StateTraceFifo.INSERT(pFIFO := pStateTraceBuffer, in := StateTimeStamp);
ELSE
	FirstEntry := FALSE;
END_IF

END_FUNCTION_BLOCK

// ---- POUs/Stn100/Stn100_10_Main.TcPOU
PROGRAM Stn100_10_Main
VAR PERSISTENT
	iStdVelocity: REAL; (*0 to 100%*)
END_VAR

VAR
	pCmp: POINTER TO udtCmpBasemain;
	pStation: POINTER TO Station;
	pStats: POINTER TO Component_Stats;
	Local: FrameworkLocal;
	Framework: FB_Framework;
	TempEvent: StatsEvent;
	pCoolingConveyor: POINTER TO udtCmpVFD;
	pVibratoryConveyor: POINTER TO udtCmpVFD;
	pVibrator: POINTER TO udtCmpVFD;
	tmrCycleAuto: TON;
	Ok2Fill: BOOL;
	bOk2Fill: BOOL;
	BoxFillComplete :BOOL;	
	tmrStarved: TON;
	Starved: BOOL;
	tmrBlocked: TON;
	Blocked: BOOL;
	TempInMoldDrop: REAL;
	TempInChuteDrop: REAL;
	tempCalc1:REAL;
	tempCalc2 : REAL;
	tempChuteCalc1 : REAL;
	tempChuteCalc2 : REAL;
	bNewBoxIndexing :BOOL;
	tmr_DelayLast : TON;

	(*Inputs*)
	iBoxPres_Infeeed AT %I*  : BOOL;
	iBoxPres_InfeedEntrance AT %I* :BOOL;
	iBoxPres_Filling AT %I*  : BOOL;
	iBoxPres_OutFeed AT %I*  : BOOL;
	iBoxPres_OutFeedExit AT %I* :BOOL;
	iWR_FillCmp AT %I* :BOOL;
	iBoxCyl_US_Retd AT%I* :BOOL;
	iBoxCyl_DS_Retd AT%I* :BOOL;
	iTempAtMoldDrop AT %I* :DINT;
	iTempAtShuteDrop AT %I* :DINT;
	iWeighRightAutoMode :BOOL;
	
	(*Sensors*)
	senBoxPresentInfeed_Entrance: FB_Sensor;
	senBoxPresentInfeed: FB_Sensor;
	senBoxPresentFilling: FB_Sensor;
	senBoxPresentOutFeed: FB_Sensor;
	senBoxPresentOutFeed_Exit: FB_Sensor;
	senWR_FillCmp: FB_SENSOR;
	senBoxCyl_US_Retd: FB_Sensor;
	senBoxCyl_DS_Retd: FB_Sensor;	
	
	(*Outputs*)
	oInfeedConv_PwrOn AT %Q* :BOOL;
	oInfeedConv_Release AT %Q* : BOOL;
	oInfeedConv_EntRelease AT %Q* : BOOL;
	oBoxCyl_US_Ret AT %Q* : BOOL;
	oBoxCyl_DS_Ret AT %Q* : BOOL;		
	oWeighRight_Start AT %Q* : BOOL;
	oWeighRight_Ok2Fill AT %Q* : BOOL;	
	oOutFeedConv_PwrOn AT %Q* :BOOL;	
	oOutFeedConv_Recieve AT %Q* :BOOL;	
	oOutFeedConv_ExitRelease AT %Q* :BOOL;
	
	(*Operator Inputs*)
	hiBoxCylExt: BOOL;
	hiBoxCylRet: BOOL;	
	hiInfeedBox_Release : BOOL;
	hoActTempMoldDrop : LREAL;
	hoActTempShuteDrop : LREAL;
	hiInfeedReleaseEntrance : BOOL;
	hiInfeedReleaseExit : BOOL;
	hiOutfeedReleaseEntrance : BOOL;
	hiOutfeedReleaseExit : BOOL;
	hoBoxPrintReq :BOOL;
	hiBoxPrintAck :BOOL;
	

END_VAR

IF Globals.gFirstScan THEN
	pCmp := ADR(Globals.gStn100_10_Main);
	pStation := ADR(Globals.gStation100);
	pStats :=ADR(Globals.gStn100_02_Stats);
	(*Address your components here that are owned by this Main*)
	pCoolingConveyor := ADR(Globals.gStn100_20_CoolingConveyor);
	pVibratoryConveyor := ADR(Globals.gStn100_30_VibratoryConveyor);
	pVibrator := ADR(Globals.gStn100_40_Vibrator);

	Local.Name :=pCmp^.Framework.ComponentIDRecord.Name;
	Local.pStateTraceBuffer := ADR(Globals.gStn100_StateTraceBuffer);
	Local.pStateTraceFifo := ADR(Globals.gStn100_StateTraceFifo);
	Local.pStats := ADR(Globals.gStn100_02_Stats);
	Local.FaultTimeLong := T#10000MS;
	Local.FaultTimeShort := T#5000MS;
	
	DefineMessages();
END_IF

FrameWork(pFramework := ADR(pCmp^.Framework), 
		  pLocal := ADR(Local), 
		  pStation := pStation);

(*House Keeping*)
Ok2Fill:=(senBoxPresentFilling.ON AND bOk2Fill);
BoxFillComplete :=(senWR_FillCmp.ON);
iWeighRightAutoMode := Globals.gWeighRightInputs.2;
oWeighRight_Ok2Fill := (Ok2Fill AND Local.CycleAuto);


(*Sensor debounce*)
senBoxPresentInfeed_Entrance(Input := iBoxPres_InfeedEntrance, DelayON := T#100MS, DelayOFF := T#100MS);
senBoxPresentInfeed(Input := iBoxPres_Infeeed, DelayON := T#100MS, DelayOFF := T#100MS);
senBoxPresentFilling(Input := iBoxPres_Filling, DelayON := T#2500MS, DelayOFF := T#100MS);
senBoxPresentOutFeed(Input := iBoxPres_OutFeed, DelayON := T#100MS, DelayOFF := T#100MS);
senBoxPresentOutFeed_Exit(Input := iBoxPres_OutFeedExit, DelayON := T#100MS, DelayOFF := T#100MS);
senWR_FillCmp(Input := iWR_FillCmp, DelayON := T#300MS, DelayOFF := T#300MS);
senBoxCyl_US_Retd(Input := iBoxCyl_US_Retd, DelayON := T#300MS, DelayOFF := T#300MS);
senBoxCyl_DS_Retd(Input := iBoxCyl_DS_Retd, DelayON := T#300MS, DelayOFF := T#300MS);

(*Set base speed reference for all sorting components*)
pCoolingConveyor^.BaseSpeedRef := iStdVelocity;
pVibratoryConveyor^.BaseSpeedRef := iStdVelocity;
pVibrator^.BaseSpeedRef := iStdVelocity;
(*Calc Degrees F from Inputs*)
TempInMoldDrop :=DINT_TO_REAL(iTempAtMoldDrop)/100;
tempCalc1 :=((TempInMoldDrop*9/5));
tempCalc2 := tempCalc1 +32.0;
hoActTempMoldDrop :=REAL_TO_LREAL(tempCalc2);
TempInChuteDrop :=DINT_TO_REAL(iTempAtShuteDrop)/100;
tempChuteCalc1 :=((TempInChuteDrop*9/5));
tempChuteCalc2 := tempChuteCalc1 +32.0;
hoActTempShuteDrop :=REAL_TO_LREAL(tempChuteCalc2);

(*Retract the BoxHold Down Cyl on an emergency stop*)
IF pStation^.EmergencyStop THEN
	(*oBoxCylRet := FALSE;*)
END_IF
(* Boxes Not Present Conditions*)
tmrStarved(IN:=(Local.CycleAuto AND Local.State = 0 AND NOT iBoxPres_Infeeed), PT:=T#1S);
tmrBlocked(IN:=(Local.CycleAuto AND Local.State = 0 AND iBoxPres_OutFeed), PT:=T#1S);
(* HACK Alert Added this Delay to allow last dump to settle*)
tmr_DelayLast(IN:=Local.State = 100, PT:=T#6S);	

IF NOT Starved AND tmrStarved.Q THEN
	Starved := TRUE;
	TempEvent.EType := Globals.cStats.Starved;
	F_SendEvent(ADR(pStats^.StatsEventFIFO),ADR(pStats^.StatsEventBuffer),ADR(TempEvent));
END_IF
IF Starved AND Local.State <> 0 THEN
	Starved := FALSE;
	IF Local.CycleAuto THEN
		TempEvent.EType := Globals.cStats.Working;
		F_SendEvent (ADR(pStats^.StatsEventFIFO), ADR(pStats^.StatsEventBuffer), ADR(TempEvent));
	END_IF
END_IF

IF NOT Blocked AND tmrBlocked.Q THEN
	Blocked := TRUE;
	TempEvent.EType := Globals.cStats.Blocked;
	F_SendEvent(ADR(pStats^.StatsEventFIFO),ADR(pStats^.StatsEventBuffer),ADR(TempEvent));
END_IF
IF Blocked AND Local.State <> 0 THEN
	Blocked := FALSE;
	IF Local.CycleAuto THEN
		TempEvent.EType := Globals.cStats.Working;
		F_SendEvent (ADR(pStats^.StatsEventFIFO), ADR(pStats^.StatsEventBuffer), ADR(TempEvent));
	END_IF
END_IF


(**********************
    Sequence logic
***********************)
CASE Local.State OF
	
0: (*Wait for Something to Do*)		
	Local.OKToStop := TRUE;
	oInfeedConv_PwrOn := TRUE;
	oOutFeedConv_PwrOn := TRUE;
	
	IF NOT pStation^.StopRequest AND((NOT pCoolingConveyor^.Running AND Ok2Fill) AND NOT(BoxFillComplete)) THEN
		Local.NextState := 10;
	END_IF
	
	IF NOT(senBoxPresentFilling.ON)AND(senBoxPresentInfeed.ON) AND NOT (bNewBoxIndexing) THEN
		Local.NextState := 50;
	END_IF
	
	IF(senBoxPresentInfeed_Entrance.ON AND NOT senBoxPresentInfeed.ON)  AND (Ok2Fill) THEN
		Local.NextState :=200;
	END_IF
	
	//IF(senBoxPresentOutFeed.ON AND NOT senBoxPresentOutFeed_Exit.ON) THEN
	//	Local.NextState :=300;
	//END_IF	
	
	IF(BoxFillComplete) AND (senBoxPresentFilling.ON) AND NOT(senBoxPresentOutFeed.ON AND senBoxPresentOutFeed_Exit.ON) THEN
		Local.NextState := 100;
	END_IF
	(* Wait For The Exit Area Clear Before Proceeding Prompt Operator*)
	IF (BoxFillComplete) AND (senBoxPresentFilling.ON) AND (senBoxPresentOutFeed.ON OR senBoxPresentOutFeed_Exit.ON) THEN
		
		Local.NextState := 5;
	END_IF
	
10: (*Start the Cooling Conveyor*)
	IF Local.FirstEntry THEN
		pCoolingConveyor^.RunReq :=TRUE;
	END_IF	
	
	Local.OKToStop := TRUE;	
	
	(*Wait for the Cooling Conveyor Running Signal*)
	IF pCoolingConveyor^.Running THEN
		Local.NextState := 20;
	END_IF
	
20: (*Start the Vibrator*)
	IF Local.FirstEntry THEN
		pVibrator^.RunReq :=TRUE;
	END_IF	
	
	Local.OKToStop := TRUE;	
	
	(*Wait for the Vibrator Running Signal*)
	IF pVibrator^.Running THEN
		oWeighRight_Ok2Fill :=TRUE;
		oWeighRight_Start :=TRUE;
		bOk2Fill := TRUE;
		Local.NextState := 0;
	END_IF	

50: (*Index Box into Filling Area*)
	IF Local.FirstEntry THEN
		pVibratoryConveyor^.RunReq :=1;
	END_IF
	
	Local.OKToStop := FALSE;
	
	IF (pVibratoryConveyor^.Running) THEN
		Local.NextState := 60;
	END_IF
	
60: (*Fillig Conv Running Release BOX from Infeed*)
	IF Local.FirstEntry THEN
		oBoxCyl_US_Ret :=FALSE;
		oBoxCyl_DS_Ret :=TRUE;
		Local.tmrFault.PT :=T#2000MS;
	END_IF
		Local.OKToStop := TRUE; 
		
	IF NOT(senBoxCyl_US_Retd.ON) AND (senBoxCyl_DS_Retd.ON)THEN
		Local.NextState := 65;
	END_IF
	
	IF Local.tmrFault.Q THEN
		IF (senBoxCyl_US_Retd.ON) THEN
			Local.FaultNumber :=1;
		END_IF
		IF NOT(senBoxCyl_DS_Retd.ON) THEN
			Local.FaultNumber :=2;
		END_IF		
	END_IF

65: (* Wait Box Present*)
	Local.OKToStop := TRUE;
	IF Local.FirstEntry THEN
		oInfeedConv_Release	:=TRUE;
		bNewBoxIndexing :=TRUE;
	END_IF	

	IF NOT (senBoxPresentInfeed.ON) THEN
		oInfeedConv_Release	:=FALSE;
	END_IF
	IF (senBoxPresentFilling.ON) THEN
		oInfeedConv_Release	:=FALSE;
		Local.NextState := 70;
	END_IF		
70: (*Stop the Conv and Ext Cylinder*)
	Local.OKToStop := TRUE;
	IF Local.FirstEntry THEN
		pVibratoryConveyor^.RunReq :=0;
	END_IF
	
	IF NOT pVibratoryConveyor^.Running  THEN
		Local.NextState := 80;
	END_IF

80: (*Ext Box Cylinder*)
	Local.OKToStop := TRUE;
	IF Local.FirstEntry THEN
		oBoxCyl_DS_Ret :=FALSE;
	END_IF
	
	IF NOT(senBoxCyl_DS_Retd.ON) THEN
		Local.NextState := 0;
		bNewBoxIndexing :=FALSE;
		bOk2Fill :=TRUE;
	END_IF

100: (*Box Fill Complete Release Full and Allow Empty*)
	(*Retract Hold Down Cylinder*)
	IF Local.FirstEntry THEN
		(**)
	END_IF
		Local.LongFaultState :=TRUE;
		Local.OKToStop := (tmr_DelayLast.Q);
		
	IF(tmr_DelayLast.Q) THEN	
		pCoolingConveyor^.RunReq :=FALSE;
		pVibrator^.RunReq :=FALSE;
		oWeighRight_Start :=FALSE;
		oBoxCyl_US_Ret :=TRUE;		
	END_IF
	
	IF (senBoxCyl_US_Retd.ON) THEN
		Local.NextState := 110;
		Local.LongFaultState :=FALSE;
	END_IF

110: (*Check Exit Area for Box Present*)
		Local.OKToStop := TRUE;			
	IF (Local.FirstEntry) THEN
		TempEvent.EType := Globals.cStats.Good;
		TempEvent.Data[0] := 1500;
		F_SendEvent(ADR(pStats^.StatsEventFIFO),ADR(pStats^.StatsEventBuffer),ADR(TempEvent));

	END_IF
	
	IF NOT(senBoxPresentOutFeed.ON) THEN
		hoBoxPrintReq :=TRUE;
		Local.NextState :=115;
	END_IF
	
115: (* Retract DS Cylinder*)
		Local.OKToStop := TRUE;	
		IF Local.FirstEntry THEN
			oBoxCyl_DS_Ret :=FALSE;
		END_IF

	IF NOT(senBoxCyl_DS_Retd.ON) THEN
		Local.NextState :=120;
	END_IF

120: (*Release Box From Filling Area*)
	IF Local.FirstEntry THEN
		bOk2Fill := FALSE;
		pVibratoryConveyor^.RunReq :=TRUE;
		oOutFeedConv_Recieve :=TRUE;	
	END_IF
	
	Local.OKToStop := TRUE;	
	(*Wait for the Box to Arrive at the Outfeed Conv*)
	IF (senBoxPresentOutFeed.ON) OR (senBoxPresentOutFeed_Exit.ON) THEN
		oOutFeedConv_Recieve :=FALSE;
		Local.NextState :=130;
	END_IF
	
130: (* Check *)
	Local.OKToStop := TRUE;
		IF Local.FirstEntry THEN
			(* *)
		END_IF
		
	(*Wzit for Box Not Present at Filling*)
	IF NOT(senBoxPresentFilling.ON) THEN
		Local.NextState :=0;
	END_IF	

200: (*Box Infeed Entrance Present and No Box Present for Loading*)
	IF Local.FirstEntry THEN
		oInfeedConv_EntRelease := TRUE;
		oInfeedConv_Release :=TRUE;	
	END_IF
	
	IF (senBoxPresentInfeed.ON) THEN
		Local.NextState :=0;
		oInfeedConv_EntRelease := FALSE;
		oInfeedConv_Release :=FALSE;			
	END_IF
	
300: (*Box OutFeed Present at Loading and Nothing Present at Exit Index The Box*)
	IF Local.FirstEntry THEN
		oOutFeedConv_Recieve := TRUE;
		oOutFeedConv_ExitRelease :=TRUE;	
	END_IF
	
	IF (senBoxPresentOutFeed_Exit.ON) THEN
		Local.NextState :=0;
		oOutFeedConv_Recieve := FALSE;
		oOutFeedConv_ExitRelease :=FALSE;			
	END_IF
(**********************
    Idle and Reset logic
***********************)
5000: (*Idle*)
	IF Local.FirstEntry THEN
		(*If this component owns components, reset the ResetStart flags here*)
		pCmp^.Framework.ResetDone := FALSE;
		Local.ManualCycleDone := FALSE;
		pCoolingConveyor^.Framework.ResetStart := 0;
		pVibratoryConveyor^.Framework.ResetStart := 0;
		pVibrator^.Framework.ResetStart := 0;
		oWeighRight_Ok2Fill :=FALSE;
		oWeighRight_Start :=FALSE;
		oInfeedConv_PwrOn := FALSE;
		oInfeedConv_Release :=FALSE;
		oInfeedConv_EntRelease :=FALSE;
		oOutFeedConv_PwrOn := FALSE;
		oOutFeedConv_Recieve :=FALSE;
		oOutFeedConv_ExitRelease :=FALSE;
		pVibratoryConveyor^.RunReq :=0;
		Local.ReEntryState := 0; 
		bNewBoxIndexing :=0;
	END_IF
	
